	10://Clear old Data on GVL 	
		Lynus_Standards.GVL_Energy.stDataHeatingPumps[diNrOfEMS_IN_CP,diNrOfHP_OUT].bEnabled := FALSE;
			Lynus_Standards.GVL_Energy.stDataHeatingPumps[diNrOfEMS_IN_CP,diNrOfHP_OUT].arrMaxPower[1] := 0;
				Lynus_Standards.GVL_Energy.stDataHeatingPumps[diNrOfEMS_IN_CP,diNrOfHP_OUT].arrMaxPower[2] := 0;
					Lynus_Standards.GVL_Energy.stDataHeatingPumps[diNrOfEMS_IN_CP,diNrOfHP_OUT].bIsControllable := FALSE;
						Lynus_Standards.GVL_Energy.stDataHeatingPumps[diNrOfEMS_IN_CP,diNrOfHP_OUT].bIsStepSwitched := FALSE;
							Lynus_Standards.GVL_Energy.stDataHeatingPumps[diNrOfEMS_IN_CP,diNrOfHP_OUT].byErrorWarning := 0;
								Lynus_Standards.GVL_Energy.stDataHeatingPumps[diNrOfEMS_IN_CP,diNrOfHP_OUT].byNumberOfSteps := 0;
									Lynus_Standards.GVL_Energy.stDataHeatingPumps[diNrOfEMS_IN_CP,diNrOfHP_OUT].byPriority := 0;
										Lynus_Standards.GVL_Energy.stDataHeatingPumps[diNrOfEMS_IN_CP,diNrOfHP_OUT].lrElPower := 0;
											Lynus_Standards.GVL_Energy.stDataHeatingPumps[diNrOfEMS_IN_CP,diNrOfHP_OUT].lrElPowerConsumption := 0;
												Lynus_Standards.GVL_Energy.stDataHeatingPumps[diNrOfEMS_IN_CP,diNrOfHP_OUT].lrElPowerProduction := 0;
													Lynus_Standards.GVL_Energy.stDataHeatingPumps[diNrOfEMS_IN_CP,diNrOfHP_OUT].rBoilerTempHeatingSys := 0;
														Lynus_Standards.GVL_Energy.stDataHeatingPumps[diNrOfEMS_IN_CP,diNrOfHP_OUT].rBoilerTempServiceWater := 0;
															Lynus_Standards.GVL_Energy.stDataHeatingPumps[diNrOfEMS_IN_CP,diNrOfHP_OUT].rFlowTemp := 0;
																Lynus_Standards.GVL_Energy.stDataHeatingPumps[diNrOfEMS_IN_CP,diNrOfHP_OUT].rFlowTempEnergySource := 0;
																	Lynus_Standards.GVL_Energy.stDataHeatingPumps[diNrOfEMS_IN_CP,diNrOfHP_OUT].rReturnTemp := 0;
																		Lynus_Standards.GVL_Energy.stDataHeatingPumps[diNrOfEMS_IN_CP,diNrOfHP_OUT].rReturnTempEnergySource := 0;										
		diNrOfEMS_IN_CP := diNrOfEMS_IN;
			//Back to the init step
			iStateGVLData := 0;

END_CASE 	 

IF diNrOfHP_OUT > 0 AND fbNumberDevice.bNumberIsCalculatet AND diNrOfEMS_IN > 0 THEN
	Lynus_Standards.GVL_Energy.stDataHeatingPumps[diNrOfEMS_IN,diNrOfHP_OUT].bEnabled := fbHP.stDataHPOut.bEnabled;
		Lynus_Standards.GVL_Energy.stDataHeatingPumps[diNrOfEMS_IN,diNrOfHP_OUT].arrMaxPower[1] := fbHP.stDataHPOut.arrMaxPower[1];
			Lynus_Standards.GVL_Energy.stDataHeatingPumps[diNrOfEMS_IN,diNrOfHP_OUT].arrMaxPower[2] := fbHP.stDataHPOut.arrMaxPower[2];
				Lynus_Standards.GVL_Energy.stDataHeatingPumps[diNrOfEMS_IN,diNrOfHP_OUT].bIsControllable := TRUE;
					Lynus_Standards.GVL_Energy.stDataHeatingPumps[diNrOfEMS_IN,diNrOfHP_OUT].bIsStepSwitched := fbHP.stDataHPOut.bIsStepSwitched;
						Lynus_Standards.GVL_Energy.stDataHeatingPumps[diNrOfEMS_IN,diNrOfHP_OUT].byErrorWarning := fbHP.stDataHPOut.byErrorWarning;
							Lynus_Standards.GVL_Energy.stDataHeatingPumps[diNrOfEMS_IN,diNrOfHP_OUT].byNumberOfSteps := fbHP.stDataHPOut.byNumberOfSteps;
								Lynus_Standards.GVL_Energy.stDataHeatingPumps[diNrOfEMS_IN,diNrOfHP_OUT].byPriority := fbHP.stDataHPOut.byPriority;
									Lynus_Standards.GVL_Energy.stDataHeatingPumps[diNrOfEMS_IN,diNrOfHP_OUT].lrElPower := fbHP.stDataHPOut.lrElPower;
										Lynus_Standards.GVL_Energy.stDataHeatingPumps[diNrOfEMS_IN,diNrOfHP_OUT].lrElPowerConsumption := fbHP.stDataHPOut.lrElPowerConsumption;
											Lynus_Standards.GVL_Energy.stDataHeatingPumps[diNrOfEMS_IN,diNrOfHP_OUT].lrElPowerProduction := fbHP.stDataHPOut.lrElPowerProduction;
												Lynus_Standards.GVL_Energy.stDataHeatingPumps[diNrOfEMS_IN,diNrOfHP_OUT].rBoilerTempHeatingSys := fbHP.stDataHPOut.rBoilerTempHeatingSys;
													Lynus_Standards.GVL_Energy.stDataHeatingPumps[diNrOfEMS_IN,diNrOfHP_OUT].rBoilerTempServiceWater := fbHP.stDataHPOut.rBoilerTempServiceWater;
														Lynus_Standards.GVL_Energy.stDataHeatingPumps[diNrOfEMS_IN,diNrOfHP_OUT].rFlowTemp := fbHP.stDataHPOut.rFlowTemp;
															Lynus_Standards.GVL_Energy.stDataHeatingPumps[diNrOfEMS_IN,diNrOfHP_OUT].rFlowTempEnergySource := fbHP.stDataHPOut.rFlowTempEnergySource;
																Lynus_Standards.GVL_Energy.stDataHeatingPumps[diNrOfEMS_IN,diNrOfHP_OUT].rReturnTemp := fbHP.stDataHPOut.rReturnTemp;
																	Lynus_Standards.GVL_Energy.stDataHeatingPumps[diNrOfEMS_IN,diNrOfHP_OUT].rReturnTempEnergySource := fbHP.stDataHPOut.rReturnTempEnergySource;	
END_IF

(*----------------------------------------------------------Save persistent data----------------------------------------------------------------*)

arrPD[1](lrValue:= BOOL_TO_LREAL(bEnable), bEventBasedActive=> );
arrPD[2](lrValue:= BOOL_TO_LREAL(bPowerDataInvers), bEventBasedActive=> );
arrPD[3](lrValue:= DINT_TO_LREAL(diNrOfEMS_IN), bEventBasedActive=> );
arrPD[4](lrValue:= DINT_TO_LREAL(diNrOfEM_IN_HP), bEventBasedActive=> );
arrPD[5](lrValue:= DINT_TO_LREAL(diNrOfEMS_IN_CP), bEventBasedActive=> );
arrPD[6](lrValue:= REAL_TO_LREAL(stSetupHP.rMaxPower1), bEventBasedActive=> );
arrPD[7](lrValue:= REAL_TO_LREAL(stSetupHP.rMaxPower2), bEventBasedActive=> );
arrPD[8](lrValue:= BOOL_TO_LREAL(stSetupHP.bManualyOn), bEventBasedActive=> );
arrPD[9](lrValue:= BOOL_TO_LREAL(stSetupHP.bOnEmergPowerOff), bEventBasedActive=> );
arrPD[10](lrValue:= BOOL_TO_LREAL(stSetupHP.bOnEmergPowerOff), bEventBasedActive=> );
arrPD[11](lrValue:= BOOL_TO_LREAL(stSetupHP.bTimeEnabled), bEventBasedActive=> );
arrPD[12](lrValue:= BYTE_TO_LREAL(stSetupHP.byDisableSOC), bEventBasedActive=> );
arrPD[13](lrValue:= BYTE_TO_LREAL(stSetupHP.byEnableSOC), bEventBasedActive=> );
arrPD[14](lrValue:= BYTE_TO_LREAL(stSetupHP.byHourOff), bEventBasedActive=> );
arrPD[15](lrValue:= BYTE_TO_LREAL(stSetupHP.byHourOn), bEventBasedActive=> );
arrPD[16](lrValue:= BYTE_TO_LREAL(stSetupHP.byManualyTargetPower), bEventBasedActive=> );
arrPD[17](lrValue:= BYTE_TO_LREAL(stSetupHP.byMinutesOff), bEventBasedActive=> );
arrPD[18](lrValue:= BYTE_TO_LREAL(stSetupHP.byMinutesOn), bEventBasedActive=> );
arrPD[19](lrValue:= BYTE_TO_LREAL(stSetupHP.byPriority), bEventBasedActive=> );
arrPD[20](lrValue:= BYTE_TO_LREAL(stSetupHP.byTimeEnabledTargetPower), bEventBasedActive=> );
arrPD[21](lrValue:= BOOL_TO_LREAL(bNoLinear), bEventBasedActive=> );
arrPD[22](lrValue:= REAL_TO_LREAL(arrTableOfInterpolationPoints[1]), bEventBasedActive=> );
arrPD[23](lrValue:= REAL_TO_LREAL(arrTableOfInterpolationPoints[2]), bEventBasedActive=> );
arrPD[24](lrValue:= REAL_TO_LREAL(arrTableOfInterpolationPoints[3]), bEventBasedActive=> );
arrPD[25](lrValue:= REAL_TO_LREAL(arrTableOfInterpolationPoints[4]), bEventBasedActive=> );
arrPD[26](lrValue:= REAL_TO_LREAL(arrTableOfInterpolationPoints[5]), bEventBasedActive=> );
arrPD[27](lrValue:= REAL_TO_LREAL(arrTableOfInterpolationPoints[6]), bEventBasedActive=> );
arrPD[28](lrValue:= REAL_TO_LREAL(arrTableOfInterpolationPoints[7]), bEventBasedActive=> );
arrPD[29](lrValue:= REAL_TO_LREAL(arrTableOfInterpolationPoints[8]), bEventBasedActive=> );
arrPD[30](lrValue:= REAL_TO_LREAL(arrTableOfInterpolationPoints[9]), bEventBasedActive=> );
arrPD[31](lrValue:= REAL_TO_LREAL(arrTableOfInterpolationPoints[10]), bEventBasedActive=> );

END_FUNCTION_BLOCK

// ---- FBs/Heating Pump/SG Ready General/FB_HP_SGReady_General_2Stage.TcPOU
FUNCTION_BLOCK FB_HP_SGReady_General_2Stage
VAR_INPUT PERSISTENT
	bEnable									: BOOL;												//{#lynus.ag#()} //Enable the Fuctionblock and his logic
	bPowerDataInvers						: BOOL;												//With True its possible to invert all received power data from the electric meter
	diNrOfEMS_IN							: DINT;												//Number of EMS what control this Device.
	diNrOfEM_IN_HP							: DINT;												//Number of the electric meter for incoming power data. (Power Data for this Device)
	stSetupHP								: ST_Setup_HP;										//{#lynus.ag#()} //Setup heating pump
END_VAR
VAR_INPUT
END_VAR
VAR_OUTPUT
	stDataHP								: ST_HP_Output;										//{#lynus.ag#()} //Output Data Heating pump
	diNrOfHP_OUT							: DINT;												//Active Number from the heating pump for using on other functions	
	rTargetPowerForExtFunc					: REAL;												//Target Power from 0% to +100% to use on a external Function	
END_VAR
VAR
	{attribute 'hide'}
	fbHP									: FB_HeatingPump;									//Function block for heating pump
	{attribute 'hide'}
	fbNumberDevice							: FB_NumberOfDevice;								//Function block to calcualte the number of the Device
	fbDIExternalLock						: FB_XL1XXX_DI;										//Digital Input from external loock signal
	fbDIErrorHP								: FB_XL1XXX_DI;										//Digital Input for error from the heating pump
	fbDOSGReady1							: FB_XL2XXX_DO;										//1 Digital Output signal for SG Ready 
	fbDOSGReady2							: FB_XL2XXX_DO;										//2 Digital Output signal for SG Ready 
	{attribute 'hide'}
	timDissableFunctions					: TON;												//Timer to dissable the Function after Lynus_Standards.Constants_General.tTimeDissableLynusFunctions Days without connection to the Lynus Cloud
	{attribute 'hide'}
	timResetConnectionOnGVL					: TON;												//Timer to try reset the connection Flag on the GVL. (When somebody delete the Connection Function and make only a onlinechange)
	{attribute 'hide'}
	timGetTime								: TON;												//Timer to activate the function tho read out the windows system time
	{attribute 'hide'}
	FNReset									: F_TRIG;											//Internal negative edge
	{attribute 'hide'}
	fbGetSystemTime							: NT_GetTime;										//Function to read out the windows system time on the local plc
	{attribute 'hide'}
	arrPD									: ARRAY[1..20] OF FB_PersistentData_Number;			//Function to save persistent data
	{attribute 'hide'}
	byWaitInStep							: BYTE;												//Wait in Step before start to clean data on PLC
	{attribute 'hide'}
	iStateGVLData							: INT;												//State machine to handle the data on the GVL
	{attribute 'hide'}
	diNumberOfActiveBatterys				: DINT;												//Number of active batterys
	{attribute 'hide'}
	diNumberOfBatteryInverterInEPO			: DINT;												//Number of battery inverters that work in Emergency Power operation 
	{attribute 'hide'}
	diCounterForGVL							: DINT;												//Counter to clean old data on GVL
	{attribute 'hide'}
	diLPForGVL								: DINT;												//Loop to clean old data on GVL
	{attribute 'hide'}	
	dwSumSOC								: DWORD;											//Sum of the SOC from all batterys
	{attribute 'hide'}
	lrGridPower								: LREAL;											//Grid power in kW
	{attribute 'hide'}
	lrSizeGridConnection					: LREAL;											//Size of the complete grid connection
	{attribute 'hide'}
	liLPBatteryData							: LINT;												//Loop to check some data from batterys
	{attribute 'hide'}
	liLPInEPO								: LINT;												//Loop to check if 1 or more battery inverters build a island grid	
	{attribute 'hide'}
	liLPGridData							: LINT;												//Loop to check some grid data
END_VAR
VAR PERSISTENT
	{attribute 'conditionalshow'}
	diNrOfEMS_IN_CP							: DINT;												//Number of EMS what control this Device to compare with the original
END_VAR

//Creator : Kai Ebensperger
//Company : Lynus AG
//Date : 19.05.2021
//Version : 1.0.0.0

//With this function block its possible to control a Heating pump with the standard and general SG-Read Interface.
//SG-Ready are 2 Digital output signals to control the Heating pump in 4 modes.
//With this Function block is also possible to display the electric and thermal power from the heating pump
//Only 2-stage machines can be controlled with this FB.

//NOTE for diNr.....Designation => 
//_IN = Here Data come in from other Functions or go out to other functions about the GVL
//_OUT = Here Data go out to other functions about the GVL

(*------------------------------------------------------------Limits----------------------------------------------------------------------------------*)

diNrOfEMS_IN := LIMIT(0,diNrOfEMS_IN,Constants_Energy.diMaxNumberOfEMS);
	diNrOfEM_IN_HP := LIMIT(0,diNrOfEM_IN_HP,Constants_Energy.diMaxNumberOfElectricMeters);
			
(*------------------------------------------------------------------Power Data----------------------------------------------------------------------------*)

IF NOT bPowerDataInvers THEN
	fbHP.lrCounterEnergyT1_Consumption := Lynus_Standards.GVL_Energy.stDataElectricMeters[diNrOfEM_IN_HP].lrCounterEnergyT1_Production * 1000;
	fbHP.lrCounterEnergyT2_Consumption := Lynus_Standards.GVL_Energy.stDataElectricMeters[diNrOfEM_IN_HP].lrCounterEnergyT2_Production * 1000;
	fbHP.lrCounterEnergyT1_Production := Lynus_Standards.GVL_Energy.stDataElectricMeters[diNrOfEM_IN_HP].lrCounterEnergyT1_Consumption * 1000;
	fbHP.lrCounterEnergyT2_Production := Lynus_Standards.GVL_Energy.stDataElectricMeters[diNrOfEM_IN_HP].lrCounterEnergyT1_Consumption * 1000;
	fbHP.lrTotalCounterEnergy_Consumption := Lynus_Standards.GVL_Energy.stDataElectricMeters[diNrOfEM_IN_HP].lrTotalCounterEnergy_Production * 1000;
	fbHP.lrTotalCounterEnergy_Production := Lynus_Standards.GVL_Energy.stDataElectricMeters[diNrOfEM_IN_HP].lrTotalCounterEnergy_Consumption * 1000;
		fbHP.lrElPowerHP := (Lynus_Standards.GVL_Energy.stDataElectricMeters[diNrOfEM_IN_HP].lrPower * 1000) * - 1;
ELSE
	fbHP.lrCounterEnergyT1_Consumption := Lynus_Standards.GVL_Energy.stDataElectricMeters[diNrOfEM_IN_HP].lrCounterEnergyT1_Consumption * 1000;
	fbHP.lrCounterEnergyT2_Consumption := Lynus_Standards.GVL_Energy.stDataElectricMeters[diNrOfEM_IN_HP].lrCounterEnergyT2_Consumption * 1000;
	fbHP.lrCounterEnergyT1_Production := Lynus_Standards.GVL_Energy.stDataElectricMeters[diNrOfEM_IN_HP].lrCounterEnergyT1_Production * 1000;
	fbHP.lrCounterEnergyT2_Production := Lynus_Standards.GVL_Energy.stDataElectricMeters[diNrOfEM_IN_HP].lrCounterEnergyT2_Production * 1000;
	fbHP.lrTotalCounterEnergy_Consumption := Lynus_Standards.GVL_Energy.stDataElectricMeters[diNrOfEM_IN_HP].lrTotalCounterEnergy_Consumption * 1000;
	fbHP.lrTotalCounterEnergy_Production := Lynus_Standards.GVL_Energy.stDataElectricMeters[diNrOfEM_IN_HP].lrTotalCounterEnergy_Production * 1000;
		fbHP.lrElPowerHP := Lynus_Standards.GVL_Energy.stDataElectricMeters[diNrOfEM_IN_HP].lrPower * 1000;
END_IF

(*-------------------------------------------------------------Calcualte the number of HP---------------------------------------------------------------*)

fbNumberDevice(
	diActualNumberOfDevices:= Lynus_Standards.GVL_Energy.stNumberOfDevices.diNumberOfHP, 
	diMaxNumberOfDevices:= Constants_Energy.diMaxNumberOfHeatingPumps, 
	udiCounterOnlineChange:= TwinCAT_SystemInfoVarList._AppInfo.OnlineChangeCnt, 
	bNumberIsCalculatet=> , 
	bFPNumberIsCalculatet=> , 
	bOnlineChange=> , 
	diNumberForThisDevice=> diNrOfHP_OUT, 
	diNumberOfTotalDevices=> );

//Write new Numer on GVL
IF fbNumberDevice.bFPNumberIsCalculatet THEN
	Lynus_Standards.GVL_Energy.stNumberOfDevices.diNumberOfHP := fbNumberDevice.diNumberOfTotalDevices;	
END_IF 

//Delete old Number on GVL
IF fbNumberDevice.bOnlineChange THEN 
	Lynus_Standards.GVL_Energy.stNumberOfDevices.diNumberOfHP := diNrOfHP_OUT;	
		iStateGVLData := 1; 
END_IF

(*-------------------------------------------------------------Get the local windows system time for this plc---------------------------------------------------------------*)
timGetTime(IN:= bEnable AND NOT timGetTime.Q, PT:= T#30S, Q=> , ET=> );

fbGetSystemTime(
	NETID:= , 
	START:= timGetTime.Q AND NOT fbGetSystemTime.BUSY, 
	TMOUT:= , 
	BUSY=> , 
	ERR=> , 
	ERRID=> , 
	TIMESTR=> );	

fbHP.stSystemTime.wHour := fbGetSystemTime.TIMESTR.wHour;
	fbHP.stSystemTime.wMinute := fbGetSystemTime.TIMESTR.wMinute;	

(*-------------------------------------------------------------Service from Backend is ready and check the connection to backen for dissabel/enable Function---------------------------------------------------------------*)

//Try to reset the variable for connection on the GVL. When all is normal then the Lynus Mqtt connection function set this variable to true in the next cycle
//When we have no connection to the backend then after Lynus_Standards.Constants_General.tTimeDissableLynusFunctions days the Function is dissabled with all of his functionalities
timResetConnectionOnGVL(IN:= NOT timResetConnectionOnGVL.Q, PT:= T#1H, Q=> , ET=> );
	IF timResetConnectionOnGVL.Q THEN Lynus_Standards.GVL_Communicator.bStateConnectionToEnableFunctions := FALSE; END_IF
		IF NOT Lynus_Standards.GVL_Communicator.bStateConnectionToEnableFunctions THEN timDissableFunctions.IN := TRUE; ELSE timDissableFunctions.IN := FALSE; END_IF  
			timDissableFunctions(IN:= , PT:= Lynus_Standards.Constants_General.tTimeDissableLynusFunctions, Q=> , ET=> );		
	
(*------------------------------------------------------------------Error and Reset----------------------------------------------------------------------------*)	

fbDIErrorHP(bInvers:= FALSE, bSignal=> );

IF timDissableFunctions.Q THEN fbHP.bWarning := TRUE; fbHP.iWarningCode := 0; ELSE fbHP.bWarning := FALSE; END_IF 	
	IF Lynus_Standards.GVL_Energy.stNumberOfDevices.diNumberOfHP > Constants_Energy.diMaxNumberOfHeatingPumps OR fbDIErrorHP.bSignal OR fbGetSystemTime.ERR THEN fbHP.bError := TRUE; ELSE fbHP.bError := FALSE; END_IF 

IF Lynus_Standards.GVL_Energy.stNumberOfDevices.diNumberOfHP > Constants_Energy.diMaxNumberOfHeatingPumps THEN fbHP.iErrorCode := 1;
ELSIF fbGetSystemTime.ERR THEN fbHP.iErrorCode := 2; 
ELSIF fbDIErrorHP.bSignal THEN fbHP.iErrorCode := 0;
END_IF

FNReset(CLK:= fbHP.stDataHPOut.bSReset, Q=> );

(*------------------------------------------------------------------Logic----------------------------------------------------------------------------*)

//Calcualte the total SOC if we have more then 1 battery in our system
diNumberOfActiveBatterys := 0;
	dwSumSOC := 0;
		FOR liLPBatteryData := 1 TO Constants_Energy.diMaxNumberOfBatterys BY 1 DO
			IF Lynus_Standards.GVL_Energy.stDataOfBatterys[diNrOfEMS_IN,liLPBatteryData].bEnabled THEN diNumberOfActiveBatterys := diNumberOfActiveBatterys + 1; END_IF
				dwSumSOC := dwSumSOC + Lynus_Standards.GVL_Energy.stDataOfBatterys[diNrOfEMS_IN,liLPBatteryData].dwSOC;
		END_FOR
	
IF diNumberOfActiveBatterys > 0 THEN
	fbHP.dwBatterySOC := DINT_TO_DWORD(DWORD_TO_DINT(dwSumSOC) / diNumberOfActiveBatterys);
ELSE
	fbHP.dwBatterySOC := 100;	//When we have no battery in the ems system
END_IF

//Check if one or more Batterysystems or batteryinverter make island mode
diNumberOfBatteryInverterInEPO := 0;
	FOR liLPInEPO := 1 TO Constants_Energy.diMaxNumberOfBatteryInverters BY 1 DO
		IF Lynus_Standards.GVL_Energy.stDataOfBatteryInverters[diNrOfEMS_IN,liLPInEPO].bWorkOnIslandMode THEN fbHP.bEPOIsActive := TRUE; diNumberOfBatteryInverterInEPO := diNumberOfBatteryInverterInEPO + 1; END_IF
	END_FOR 
		IF diNumberOfBatteryInverterInEPO <= 0 THEN fbHP.bEPOIsActive := FALSE; END_IF

//Check the max. power of the grid connection and the sum of grid power
lrSizeGridConnection := 0;
	lrGridPower := 0;
		FOR liLPGridData := 1 TO Constants_Energy.diMaxNumberOfGridConnections BY 1 DO
			lrSizeGridConnection := lrSizeGridConnection + Lynus_Standards.GVL_Energy.stDataGridConnections[diNrOfEMS_IN,liLPGridData].rSizeGridConn;
				lrGridPower := lrGridPower + Lynus_Standards.GVL_Energy.stDataGridConnections[diNrOfEMS_IN,liLPGridData].lrPower;
		END_FOR		

//Feedback for HP is running
IF fbHP.arrTargetPower[1] > 0 OR fbHP.arrTargetPower[2] > 0 THEN fbHP.bHPIsRunning := TRUE; ELSE fbHP.bHPIsRunning := FALSE; END_IF 
		
//Digital input for external lock signal
fbDIExternalLock(bInvers:= FALSE, bSignal=> );

//Functionblock HP
fbHP(
	bEnable:= bEnable AND NOT timDissableFunctions.Q,  
	bError:= , 
	bWarning:= , 
	bIsStepSwitched:= TRUE, 
	bEPOIsActive:= , 
	bExternalLock:= fbDIExternalLock.bSignal, 
	bReset:= FNReset.Q, 
	bExternalOnCommand:= Lynus_Standards.GVL_Energy.stDataHeatingPumps[diNrOfEMS_IN,diNrOfHP_OUT].bExternalOnCommand, 
	bWriteWithDelay:= TRUE,
	bHPIsRunning:= , 
	iErrorCode:= , 
	iWarningCode:= , 
	dwBatterySOC:= , 
	diNumberOfHP:= diNrOfHP_OUT, 
	rBoilerTempHeatingSys:= 0, 
	rBoilerTempServiceWater:= 0, 
	rFlowTemp:= 0, 
	rReturnTemp:= 0, 
	rFlowTempEnergySource:= 0, 
	rReturnTempEnergySource:= 0, 
	lrSizeGridConnection:= lrSizeGridConnection, 
	lrGridPower:= lrGridPower, 
	lrTotalCounterEnergy_Consumption:= , 
	lrTotalCounterEnergy_Production:= , 
	lrCounterEnergyT1_Consumption:= , 
	lrCounterEnergyT2_Consumption:= , 
	lrCounterEnergyT1_Production:= , 
	lrCounterEnergyT2_Production:= , 
	lrCounterThermalEnergy_Heating:= 0, 
	lrCounterThermalEnergy_Water:= 0, 
	lrElPowerHP:= , 
	arrTargetPower:= Lynus_Standards.GVL_Energy.stDataHeatingPumps[diNrOfEMS_IN,diNrOfHP_OUT].arrTargetPowerEMS, 
	tOnDelayExternalOn:= T#2M, 
	tOffDelayExternalOn:= T#2H, 
	tMinOnTime:= T#1.5H,
	tTimDelayOutput:= T#5S, 
	stSystemTime:= , 
	stSetupHP:= stSetupHP, 
	stDataHPOut=> , 
	stDataHPOutDelay=> stDataHP, 
	arrPercentValuesSteps=> );

//Target Power, to use this on a external Function
rTargetPowerForExtFunc := fbHP.stDataHPOut.rTargetPower;
	
(*-------------------------------------------------------------------------Output----------------------------------------------------------------------*)

//Operating Mode (When Manualy mode is active)
IF stSetupHP.bManualyOn THEN	
	//Operating Mode 1 SG Ready
	IF NOT fbHP.stDataHPOut.bOutput THEN 
		fbDOSGReady1.bSignal := FALSE; 
		fbDOSGReady2.bSignal := TRUE; 
	END_IF
		//Operating Mode 2 SG Ready
		IF fbHP.stDataHPOut.rTargetPower < fbHP.arrPercentValuesSteps[1] AND fbHP.stDataHPOut.rTargetPower > 0 THEN 
			fbDOSGReady1.bSignal := FALSE; 
			fbDOSGReady2.bSignal := FALSE; 
		END_IF
			//Operating Mode 3 SG Ready
			IF fbHP.stDataHPOut.rTargetPower >= fbHP.arrPercentValuesSteps[1] AND fbHP.arrPercentValuesSteps[1] > 0 THEN 
				fbDOSGReady1.bSignal := TRUE; 
				fbDOSGReady2.bSignal := FALSE;
			END_IF
				//Operating Mode 4 SG Ready	
				IF fbHP.stDataHPOut.rTargetPower >= 100 AND fbHP.stDataHPOut.byNumberOfSteps > 1 THEN 
					fbDOSGReady1.bSignal := TRUE; 
					fbDOSGReady2.bSignal := TRUE; 
				END_IF
ELSE
	//Operating Mode (When Normal mode is active) 
	//Operating Mode 1 SG Ready
	IF NOT fbHP.stDataHPOut.bOutput THEN
		fbDOSGReady1.bSignal := FALSE; 
		fbDOSGReady2.bSignal := TRUE;
	ELSE
		//Operating Mode 2 SG Ready
		IF fbHP.stDataHPOut.bOutput THEN 
			fbDOSGReady1.bSignal := FALSE; 
			fbDOSGReady2.bSignal := FALSE; 
		END_IF
			//Operating Mode 3 SG Ready
			IF fbHP.stDataHPOut.rTargetPower >= fbHP.arrPercentValuesSteps[1] AND fbHP.arrPercentValuesSteps[1] > 0 THEN 
				fbDOSGReady1.bSignal := TRUE; 
				fbDOSGReady2.bSignal := FALSE; 
			END_IF
				//Operating Mode 4 SG Ready	
				IF fbHP.stDataHPOut.rTargetPower >= 100 AND fbHP.stDataHPOut.byNumberOfSteps > 1 THEN 
					fbDOSGReady1.bSignal := TRUE; 
					fbDOSGReady2.bSignal := TRUE;
				END_IF
	END_IF	
END_IF

fbDOSGReady1(bInvers:= FALSE, bSignal:= );
	fbDOSGReady2(bInvers:= FALSE, bSignal:= );

(*-----------------------------------------------------------Handle data to Global structure for the heating pump-----------------------------------------------------------------*)

//Delte al old Data on GVL after a online change or change on the variable diNrOfEMS_IDOD
IF diNrOfEMS_IN <> diNrOfEMS_IN_CP AND iStateGVLData = 0 THEN iStateGVLData := 10; END_IF 

CASE iStateGVLData OF
	
	0://Init Step
		byWaitInStep := 0;
			diCounterForGVL := 1;
	
	1://Wait for 4 Steps before clean al Data on GVL
		byWaitInStep := byWaitInStep + 1;
			IF byWaitInStep >= 4 AND fbNumberDevice.bNumberIsCalculatet THEN iStateGVLData := 2; END_IF
				//To much Devices, back to the Init step
				IF byWaitInStep >= 4 AND NOT fbNumberDevice.bNumberIsCalculatet THEN iStateGVLData := 0; END_IF	
			
	2://Clear all Data in GVL
		FOR diLPForGVL := 1 TO Constants_Energy.diMaxNumberOfEMS BY 1 DO
			Lynus_Standards.GVL_Energy.stDataHeatingPumps[diLPForGVL,diCounterForGVL].bEnabled := FALSE;
				Lynus_Standards.GVL_Energy.stDataHeatingPumps[diLPForGVL,diCounterForGVL].arrMaxPower[1] := 0;
					Lynus_Standards.GVL_Energy.stDataHeatingPumps[diLPForGVL,diCounterForGVL].arrMaxPower[2] := 0;
						Lynus_Standards.GVL_Energy.stDataHeatingPumps[diLPForGVL,diCounterForGVL].bIsControllable := FALSE;
							Lynus_Standards.GVL_Energy.stDataHeatingPumps[diLPForGVL,diCounterForGVL].bIsStepSwitched := FALSE;
								Lynus_Standards.GVL_Energy.stDataHeatingPumps[diLPForGVL,diCounterForGVL].byErrorWarning := 0;
									Lynus_Standards.GVL_Energy.stDataHeatingPumps[diLPForGVL,diCounterForGVL].byNumberOfSteps := 0;
										Lynus_Standards.GVL_Energy.stDataHeatingPumps[diLPForGVL,diCounterForGVL].byPriority := 0;
											Lynus_Standards.GVL_Energy.stDataHeatingPumps[diLPForGVL,diCounterForGVL].lrElPower := 0;
												Lynus_Standards.GVL_Energy.stDataHeatingPumps[diLPForGVL,diCounterForGVL].lrElPowerConsumption := 0;
													Lynus_Standards.GVL_Energy.stDataHeatingPumps[diLPForGVL,diCounterForGVL].lrElPowerProduction := 0;
														Lynus_Standards.GVL_Energy.stDataHeatingPumps[diLPForGVL,diCounterForGVL].rBoilerTempHeatingSys := 0;
															Lynus_Standards.GVL_Energy.stDataHeatingPumps[diLPForGVL,diCounterForGVL].rBoilerTempServiceWater := 0;
																Lynus_Standards.GVL_Energy.stDataHeatingPumps[diLPForGVL,diCounterForGVL].rFlowTemp := 0;
																	Lynus_Standards.GVL_Energy.stDataHeatingPumps[diLPForGVL,diCounterForGVL].rFlowTempEnergySource := 0;
																		Lynus_Standards.GVL_Energy.stDataHeatingPumps[diLPForGVL,diCounterForGVL].rReturnTemp := 0;
																			Lynus_Standards.GVL_Energy.stDataHeatingPumps[diLPForGVL,diCounterForGVL].rReturnTempEnergySource := 0;
																				//Set also the target value from ems back here to 0 and not in EMS function because EMS is in Standy when we have a online change (Problem when we delete a ems function and make a online change)
																				Lynus_Standards.GVL_Energy.stDataHeatingPumps[diLPForGVL,diCounterForGVL].arrTargetPowerEMS[1] := 0;
																					Lynus_Standards.GVL_Energy.stDataHeatingPumps[diLPForGVL,diCounterForGVL].arrTargetPowerEMS[2] := 0;
																						Lynus_Standards.GVL_Energy.stDataHeatingPumps[diLPForGVL,diCounterForGVL].bExternalOnCommand := FALSE;	
		END_FOR
			diCounterForGVL := diCounterForGVL + 1;
				diCounterForGVL := LIMIT(0,diCounterForGVL,Constants_Energy.diMaxNumberOfHeatingPumps);
					//Back to the init step
					IF diCounterForGVL >= Constants_Energy.diMaxNumberOfHeatingPumps THEN iStateGVLData := 0; END_IF

	10://Clear old Data on GVL 	
		Lynus_Standards.GVL_Energy.stDataHeatingPumps[diNrOfEMS_IN_CP,diNrOfHP_OUT].bEnabled := FALSE;
			Lynus_Standards.GVL_Energy.stDataHeatingPumps[diNrOfEMS_IN_CP,diNrOfHP_OUT].arrMaxPower[1] := 0;
				Lynus_Standards.GVL_Energy.stDataHeatingPumps[diNrOfEMS_IN_CP,diNrOfHP_OUT].arrMaxPower[2] := 0;
					Lynus_Standards.GVL_Energy.stDataHeatingPumps[diNrOfEMS_IN_CP,diNrOfHP_OUT].bIsControllable := FALSE;
						Lynus_Standards.GVL_Energy.stDataHeatingPumps[diNrOfEMS_IN_CP,diNrOfHP_OUT].bIsStepSwitched := FALSE;
							Lynus_Standards.GVL_Energy.stDataHeatingPumps[diNrOfEMS_IN_CP,diNrOfHP_OUT].byErrorWarning := 0;
								Lynus_Standards.GVL_Energy.stDataHeatingPumps[diNrOfEMS_IN_CP,diNrOfHP_OUT].byNumberOfSteps := 0;
									Lynus_Standards.GVL_Energy.stDataHeatingPumps[diNrOfEMS_IN_CP,diNrOfHP_OUT].byPriority := 0;
										Lynus_Standards.GVL_Energy.stDataHeatingPumps[diNrOfEMS_IN_CP,diNrOfHP_OUT].lrElPower := 0;
											Lynus_Standards.GVL_Energy.stDataHeatingPumps[diNrOfEMS_IN_CP,diNrOfHP_OUT].lrElPowerConsumption := 0;
												Lynus_Standards.GVL_Energy.stDataHeatingPumps[diNrOfEMS_IN_CP,diNrOfHP_OUT].lrElPowerProduction := 0;
													Lynus_Standards.GVL_Energy.stDataHeatingPumps[diNrOfEMS_IN_CP,diNrOfHP_OUT].rBoilerTempHeatingSys := 0;
														Lynus_Standards.GVL_Energy.stDataHeatingPumps[diNrOfEMS_IN_CP,diNrOfHP_OUT].rBoilerTempServiceWater := 0;
															Lynus_Standards.GVL_Energy.stDataHeatingPumps[diNrOfEMS_IN_CP,diNrOfHP_OUT].rFlowTemp := 0;
																Lynus_Standards.GVL_Energy.stDataHeatingPumps[diNrOfEMS_IN_CP,diNrOfHP_OUT].rFlowTempEnergySource := 0;
																	Lynus_Standards.GVL_Energy.stDataHeatingPumps[diNrOfEMS_IN_CP,diNrOfHP_OUT].rReturnTemp := 0;
																		Lynus_Standards.GVL_Energy.stDataHeatingPumps[diNrOfEMS_IN_CP,diNrOfHP_OUT].rReturnTempEnergySource := 0;										
		diNrOfEMS_IN_CP := diNrOfEMS_IN;
			//Back to the init step
			iStateGVLData := 0;

END_CASE 	 

IF diNrOfHP_OUT > 0 AND fbNumberDevice.bNumberIsCalculatet AND diNrOfEMS_IN > 0 THEN
	Lynus_Standards.GVL_Energy.stDataHeatingPumps[diNrOfEMS_IN,diNrOfHP_OUT].bEnabled := fbHP.stDataHPOut.bEnabled;
		Lynus_Standards.GVL_Energy.stDataHeatingPumps[diNrOfEMS_IN,diNrOfHP_OUT].arrMaxPower[1] := fbHP.stDataHPOut.arrMaxPower[1];
			Lynus_Standards.GVL_Energy.stDataHeatingPumps[diNrOfEMS_IN,diNrOfHP_OUT].arrMaxPower[2] := fbHP.stDataHPOut.arrMaxPower[2];
				Lynus_Standards.GVL_Energy.stDataHeatingPumps[diNrOfEMS_IN,diNrOfHP_OUT].bIsControllable := TRUE;
					Lynus_Standards.GVL_Energy.stDataHeatingPumps[diNrOfEMS_IN,diNrOfHP_OUT].bIsStepSwitched := fbHP.stDataHPOut.bIsStepSwitched;
						Lynus_Standards.GVL_Energy.stDataHeatingPumps[diNrOfEMS_IN,diNrOfHP_OUT].byErrorWarning := fbHP.stDataHPOut.byErrorWarning;
							Lynus_Standards.GVL_Energy.stDataHeatingPumps[diNrOfEMS_IN,diNrOfHP_OUT].byNumberOfSteps := fbHP.stDataHPOut.byNumberOfSteps;
								Lynus_Standards.GVL_Energy.stDataHeatingPumps[diNrOfEMS_IN,diNrOfHP_OUT].byPriority := fbHP.stDataHPOut.byPriority;
									Lynus_Standards.GVL_Energy.stDataHeatingPumps[diNrOfEMS_IN,diNrOfHP_OUT].lrElPower := fbHP.stDataHPOut.lrElPower;
										Lynus_Standards.GVL_Energy.stDataHeatingPumps[diNrOfEMS_IN,diNrOfHP_OUT].lrElPowerConsumption := fbHP.stDataHPOut.lrElPowerConsumption;
											Lynus_Standards.GVL_Energy.stDataHeatingPumps[diNrOfEMS_IN,diNrOfHP_OUT].lrElPowerProduction := fbHP.stDataHPOut.lrElPowerProduction;
												Lynus_Standards.GVL_Energy.stDataHeatingPumps[diNrOfEMS_IN,diNrOfHP_OUT].rBoilerTempHeatingSys := fbHP.stDataHPOut.rBoilerTempHeatingSys;
													Lynus_Standards.GVL_Energy.stDataHeatingPumps[diNrOfEMS_IN,diNrOfHP_OUT].rBoilerTempServiceWater := fbHP.stDataHPOut.rBoilerTempServiceWater;
														Lynus_Standards.GVL_Energy.stDataHeatingPumps[diNrOfEMS_IN,diNrOfHP_OUT].rFlowTemp := fbHP.stDataHPOut.rFlowTemp;
															Lynus_Standards.GVL_Energy.stDataHeatingPumps[diNrOfEMS_IN,diNrOfHP_OUT].rFlowTempEnergySource := fbHP.stDataHPOut.rFlowTempEnergySource;
																Lynus_Standards.GVL_Energy.stDataHeatingPumps[diNrOfEMS_IN,diNrOfHP_OUT].rReturnTemp := fbHP.stDataHPOut.rReturnTemp;
																	Lynus_Standards.GVL_Energy.stDataHeatingPumps[diNrOfEMS_IN,diNrOfHP_OUT].rReturnTempEnergySource := fbHP.stDataHPOut.rReturnTempEnergySource;	
END_IF

(*----------------------------------------------------------Save persistent data----------------------------------------------------------------*)

arrPD[1](lrValue:= BOOL_TO_LREAL(bEnable), bEventBasedActive=> );
arrPD[2](lrValue:= BOOL_TO_LREAL(bPowerDataInvers), bEventBasedActive=> );
arrPD[3](lrValue:= DINT_TO_LREAL(diNrOfEMS_IN), bEventBasedActive=> );
arrPD[4](lrValue:= DINT_TO_LREAL(diNrOfEM_IN_HP), bEventBasedActive=> );
arrPD[5](lrValue:= DINT_TO_LREAL(diNrOfEMS_IN_CP), bEventBasedActive=> );
arrPD[6](lrValue:= REAL_TO_LREAL(stSetupHP.rMaxPower1), bEventBasedActive=> );
arrPD[7](lrValue:= REAL_TO_LREAL(stSetupHP.rMaxPower2), bEventBasedActive=> );
arrPD[8](lrValue:= BOOL_TO_LREAL(stSetupHP.bManualyOn), bEventBasedActive=> );
arrPD[9](lrValue:= BOOL_TO_LREAL(stSetupHP.bOnEmergPowerOff), bEventBasedActive=> );
arrPD[10](lrValue:= BOOL_TO_LREAL(stSetupHP.bOnEmergPowerOff), bEventBasedActive=> );
arrPD[11](lrValue:= BOOL_TO_LREAL(stSetupHP.bTimeEnabled), bEventBasedActive=> );
arrPD[12](lrValue:= BYTE_TO_LREAL(stSetupHP.byDisableSOC), bEventBasedActive=> );
arrPD[13](lrValue:= BYTE_TO_LREAL(stSetupHP.byEnableSOC), bEventBasedActive=> );
arrPD[14](lrValue:= BYTE_TO_LREAL(stSetupHP.byHourOff), bEventBasedActive=> );
arrPD[15](lrValue:= BYTE_TO_LREAL(stSetupHP.byHourOn), bEventBasedActive=> );
arrPD[16](lrValue:= BYTE_TO_LREAL(stSetupHP.byManualyTargetPower), bEventBasedActive=> );
arrPD[17](lrValue:= BYTE_TO_LREAL(stSetupHP.byMinutesOff), bEventBasedActive=> );
arrPD[18](lrValue:= BYTE_TO_LREAL(stSetupHP.byMinutesOn), bEventBasedActive=> );
arrPD[19](lrValue:= BYTE_TO_LREAL(stSetupHP.byPriority), bEventBasedActive=> );
arrPD[20](lrValue:= BYTE_TO_LREAL(stSetupHP.byTimeEnabledTargetPower), bEventBasedActive=> );

END_FUNCTION_BLOCK

// ---- FBs/House Consumption/Virtual/FB_HouseC_Power_Virtual.TcPOU
FUNCTION_BLOCK FB_HouseC_Power_Virtual
VAR_INPUT PERSISTENT
	bEnable									: BOOL;													//{#lynus.ag#()} //Enable the Fuctionblock and his logic
	diNrOfEMS_IN							: DINT;													//Number of EMS from what this Device received Data
END_VAR
VAR_INPUT
	bSetDefault								: BOOL;													//With this Input can set the default Value from the Counter from the Input to the Counter at the Output									
	lrCounterConsumptionSetDefault			: LREAL;												//Set Default value for Consumption Counter
	lrCounterProductionSetDefault			: LREAL;												//Set Default value for Production Counter
END_VAR
VAR_OUTPUT
	stDataHouseC							: ST_HouseConsumption_Output;							//{#lynus.ag#()} //House consumption output data
	diNrOfHouseC_OUT						: DINT;													//Active Number from the House connection for using on other functions
END_VAR
VAR
	{attribute 'hide'}
	fbHouseC								: FB_HouseConsumption;									//Function for House consumption
	{attribute 'hide'}
	fbNumberDevice							: FB_NumberOfDevice;									//Function block to calcualte the number of the Device
	{attribute 'hide'}
	TaskIndex								: GETCURTASKINDEX;										//Function to read out the task index	
	{attribute 'hide'}
	timSaveCSProd							: TON;													//Timer to save the Counter Status from production on persistent data
	{attribute 'hide'}
	timSaveCSCons							: TON;													//Timer to save the Counter Status from Consumption on persistent data
	{attribute 'hide'}
	timDissableFunctions					: TON;													//Timer to dissable the Function after Lynus_Standards.Constants_General.tTimeDissableLynusFunctions Days without connection to the Lynus Cloud
	{attribute 'hide'}
	timResetConnectionOnGVL					: TON;													//Timer to try reset the connection Flag on the GVL. (When somebody delete the Connection Function and make only a onlinechange)
	{attribute 'hide'}
	FPSetDefault							: R_TRIG;												//Internal positive Edge
	{attribute 'hide'}
	arrPD									: ARRAY[1..4] OF FB_PersistentData_Number;				//Function to save persistent data 
	{attribute 'hide'}
	bError									: BOOL;													//Error from external Devices
	{attribute 'hide'}
	byWaitInStep							: BYTE;													//Wait in Step before start to clean data on PLC
	{attribute 'hide'}
	iStateGVLData							: INT;													//State machine to handle the data on the GVL
	{attribute 'hide'}
	diCounterForGVL							: DINT;													//Counter to clean old data on GVL
	{attribute 'hide'}
	udicycleTime							: UDINT;												//Cycletime of plc
	{attribute 'hide'}
	lrPowerProduction						: LREAL;												//Complete Power Production from al Devices of this EMS in kW 
	{attribute 'hide'}
	lrPowerBattery							: LREAL;												//Complete Battery Power from al Batterys of this EMS in kW 
	{attribute 'hide'}
	lrPowerGrid								: LREAL;												//Complete Grid Power from al Grids of this EMS in kW 
	{attribute 'hide'}
	lrCounterConsumption_CP					: LREAL;												//Counter Status Consumption with Unit kW/h to compare for save persistent
	{attribute 'hide'}
	lrCounterProduction_CP					: LREAL;												//Counter Status Production with Unit kW/h to compare for save persistent
	{attribute 'hide'}
	lrTotalPower							: LREAL;												//Total power with unit kW
	{attribute 'hide'}
	lrTotalPower_CP							: LREAL;												//Total power with unit kW to trigger the calculation for energy
	{attribute 'hide'}
	lrCyclesForMinute						: LREAL;												//Cycles what the plc need for 1 minute 
	{attribute 'hide'}
	lrPastTime								: LREAL;												//Past time in hours 
	{attribute 'hide'}
	lrSumToCalculate						: LREAL;												//Actual sum of the energy counters before start the calculation with unit kW/h
	{attribute 'hide'}
	liLPPower								: LINT;													//Loop to calculate the total power
END_VAR
VAR PERSISTENT
	{attribute 'conditionalshow'}
	lrCounterConsumption					: LREAL;												//Counter Status Consumption with Unit kW/h
	{attribute 'conditionalshow'}
	lrCounterProduction						: LREAL;												//Counter Status Production with Unit kW/h
END_VAR

//Creator : Kai Ebensperger
//Company : Lynus AG
//Date : 15.06.2021
//Version : 1.0.0.0

//With this function block its possible to show the power data from a house.
//The power data in this function block is calculated by all the other consumers and producers. So the output data is not messured.
//Use only one of this Function block per each EMS
//NOTE : The output from this Function Block is not 100% perfect why the value is only calculatet and not messured.

//NOTE for diNr.....Designation => 
//_IN = Here Data come in from other Functions or go out to other functions about the GVL
//_OUT = Here Data go out to other functions about the GVL

(*------------------------------------------------------------Limits----------------------------------------------------------------------------------*)

diNrOfEMS_IN := LIMIT(0,diNrOfEMS_IN,Constants_Energy.diMaxNumberOfEMS);

(*-------------------------------------------------------------Calcualte the number of House Consumption---------------------------------------------------------------*)

fbNumberDevice(
	diActualNumberOfDevices:= Lynus_Standards.GVL_Energy.stNumberOfDevices.diNumberOfHouseConsumption, 
	diMaxNumberOfDevices:= Constants_Energy.diMaxNumberOfHouseConsumptions, 
	udiCounterOnlineChange:= TwinCAT_SystemInfoVarList._AppInfo.OnlineChangeCnt, 
	bNumberIsCalculatet=> , 
	bFPNumberIsCalculatet=> , 
	bOnlineChange=> , 
	diNumberForThisDevice=> diNrOfHouseC_OUT, 
	diNumberOfTotalDevices=> );

//Write new Numer on GVL
IF fbNumberDevice.bFPNumberIsCalculatet THEN
	Lynus_Standards.GVL_Energy.stNumberOfDevices.diNumberOfHouseConsumption := fbNumberDevice.diNumberOfTotalDevices;	
END_IF 

//Delete old Number on GVL
IF fbNumberDevice.bOnlineChange THEN 
	Lynus_Standards.GVL_Energy.stNumberOfDevices.diNumberOfHouseConsumption := diNrOfHouseC_OUT;	
		iStateGVLData := 1; 
END_IF

(*-------------------------------------------------------------Calcualte the power of the house---------------------------------------------------------------*)	

lrPowerProduction := 0;
	lrPowerBattery := 0;
		lrPowerGrid := 0;
			bError := FALSE;

//Batterypower
FOR liLPPower := 1 TO Constants_Energy.diMaxNumberOfBatterys BY 1 DO
	lrPowerBattery := lrPowerBattery + Lynus_Standards.GVL_Energy.stDataOfBatterys[diNrOfEMS_IN,liLPPower].lrPower;	
		IF Lynus_Standards.GVL_Energy.stDataOfBatterys[diNrOfEMS_IN,liLPPower].byErrorWarning = 2 THEN bError := TRUE; END_IF 
END_FOR 
 	//Generator power
	FOR liLPPower := 1 TO Constants_Energy.diMaxNumberOfGenerators BY 1 DO
		lrPowerProduction := lrPowerProduction + Lynus_Standards.GVL_Energy.stDataOfGenerators[liLPPower].lrPowerProduction;	
			IF Lynus_Standards.GVL_Energy.stDataOfGenerators[liLPPower].byErrorWarning = 2 THEN bError := TRUE; END_IF		
	END_FOR 
		//PV power
		FOR liLPPower := 1 TO Constants_Energy.diMaxNumberOfPvSystems BY 1 DO
			lrPowerProduction := lrPowerProduction + Lynus_Standards.GVL_Energy.stDataOfPvSystems[liLPPower].lrPowerProduction;	
				IF Lynus_Standards.GVL_Energy.stDataOfPvSystems[liLPPower].byErrorWarning = 2 THEN bError := TRUE; END_IF		
		END_FOR	
			//Grid power	
			FOR liLPPower := 1 TO Constants_Energy.diMaxNumberOfGridConnections BY 1 DO
				lrPowerGrid := lrPowerGrid + Lynus_Standards.GVL_Energy.stDataGridConnections[diNrOfEMS_IN,liLPPower].lrPower;	
					IF Lynus_Standards.GVL_Energy.stDataGridConnections[diNrOfEMS_IN,liLPPower].byErrorWarning = 2 THEN bError := TRUE; END_IF 
			END_FOR 

//Complete power
lrTotalPower := lrPowerProduction + lrPowerGrid + lrPowerBattery;
	lrTotalPower := LIMIT(0,lrTotalPower,100000);							

(*-------------------------------------------------------------Calcualte the energy of the house---------------------------------------------------------------*)
							
//Read out the Taskindex
TaskIndex(index=> );							

//Set default Value
FPSetDefault(CLK:= bSetDefault, Q=> );
	IF FPSetDefault.Q THEN 
		lrCounterConsumption_CP := lrCounterConsumptionSetDefault;
			lrCounterProduction_CP := lrCounterProductionSetDefault;
	END_IF
						
//Save the persistent counter status to the counter status for compare on the first plc cycle	
IF TwinCAT_SystemInfoVarList._TaskInfo[TaskIndex.index].FirstCycle THEN 
	lrCounterConsumption_CP := lrCounterConsumption;
		lrCounterProduction_CP := lrCounterProduction;
END_IF											

//Timer to save the Energy Counters persistent every 12 hours											
timSaveCSProd(IN:= lrCounterProduction <> lrCounterProduction_CP, PT:= T#12H, Q=> , ET=> );
	timSaveCSCons(IN:= lrCounterConsumption <> lrCounterConsumption_CP, PT:= T#12H, Q=> , ET=> );

IF timSaveCSProd.Q THEN lrCounterProduction := lrCounterProduction_CP; END_IF 
	IF timSaveCSCons.Q THEN lrCounterConsumption := lrCounterConsumption_CP; END_IF  
	
//Write Data when the Event Based saving on persitent Data is not active
IF NOT arrPD[3].bEventBasedActive AND NOT arrPD[4].bEventBasedActive THEN
	lrCounterProduction := lrCounterProduction_CP;
		lrCounterConsumption := lrCounterConsumption_CP;
END_IF   
			
//Read out the cycle time to calculate the energy counters
//Cycle Time in MS
udicycleTime := TwinCAT_SystemInfoVarList._TaskInfo[TaskIndex.index].CycleTime / 10000;

//Calculate the cycles what is needed for 1 Minute
lrCyclesForMinute := UDINT_TO_LREAL((1 * udicycleTime)) / 60000;	

//Calculate past time in hours
lrPastTime := lrPastTime + (lrCyclesForMinute / 60);

//Calculate the Energy when the power data change and start then from new
IF MEMCMP(ADR(lrTotalPower),ADR(lrTotalPower_CP),SIZEOF(lrTotalPower_CP)) <> 0 THEN
	//INFO : Negative Value at the moment is not in use about the limitation of the Total power
	IF lrSumToCalculate < 0 THEN
		lrCounterProduction_CP := lrCounterProduction_CP + (lrSumToCalculate * - 1);
	ELSE
		lrCounterConsumption_CP := lrCounterConsumption_CP + lrSumToCalculate;
	END_IF
		lrSumToCalculate := 0;
			lrPastTime := 0;
				lrTotalPower_CP := lrTotalPower;
END_IF

//Calculate the sum after the calculation why we must calculate after the power change
lrSumToCalculate := lrTotalPower * lrPastTime;

(*-------------------------------------------------------------Service from Backend is ready and check the connection to backen for dissabel/enable Function---------------------------------------------------------------*)

//Try to reset the variable for connection on the GVL. When all is normal then the Lynus Mqtt connection function set this variable to true in the next cycle
//When we have no connection to the backend then after Lynus_Standards.Constants_General.tTimeDissableLynusFunctions days the Function is dissabled with all of his functionalities
timResetConnectionOnGVL(IN:= NOT timResetConnectionOnGVL.Q, PT:= T#1H, Q=> , ET=> );
	IF timResetConnectionOnGVL.Q THEN Lynus_Standards.GVL_Communicator.bStateConnectionToEnableFunctions := FALSE; END_IF
		IF NOT Lynus_Standards.GVL_Communicator.bStateConnectionToEnableFunctions THEN timDissableFunctions.IN := TRUE; ELSE timDissableFunctions.IN := FALSE; END_IF  
			timDissableFunctions(IN:= , PT:= Lynus_Standards.Constants_General.tTimeDissableLynusFunctions, Q=> , ET=> );

(*-----------------------------------------------------------------------------Error ----------------------------------------------------------------------------*)

IF timDissableFunctions.Q THEN fbHouseC.bWarning := TRUE; fbHouseC.iWarningCode := 0; ELSE fbHouseC.bWarning := FALSE; END_IF 	
	IF Lynus_Standards.GVL_Energy.stNumberOfDevices.diNumberOfHouseConsumption > Constants_Energy.diMaxNumberOfHouseConsumptions OR bError THEN fbHouseC.bError := TRUE; ELSE fbHouseC.bError := FALSE; END_IF 
		IF Lynus_Standards.GVL_Energy.stNumberOfDevices.diNumberOfHouseConsumption > Constants_Energy.diMaxNumberOfHouseConsumptions THEN fbHouseC.iErrorCode := 1;
		ELSIF bError THEN fbHouseC.iErrorCode := 0; 
		END_IF  

(*------------------------------------------------------------------FB House----------------------------------------------------------------------------*)	
	
fbHouseC(
	bEnable:= bEnable AND NOT timDissableFunctions.Q,
	bError:= , 
	bWriteWithDelay:= TRUE, 
	iErrorCode:= , 
	iWarningCode:= , 
	lrTotalCounterEnergy_Consumption:= lrCounterConsumption_CP * 1000, 
	lrTotalCounterEnergy_Production:= lrCounterProduction_CP * 1000, 
	lrCounterEnergyT1_Consumption:= lrCounterConsumption_CP * 1000, 
	lrCounterEnergyT2_Consumption:= , 
	lrCounterEnergyT1_Production:= lrCounterProduction_CP * 1000, 
	lrCounterEnergyT2_Production:= , 
	lrPowerHouseConsumption:= lrTotalPower * 1000, 
	tTimDelayOutput:= T#5S, 
	stDataHouseCOut=> , 
	stDataHouseCOutDelay=> stDataHouseC);
	
	(*-----------------------------------------------------------Handle data to Global structure for the House consumption-----------------------------------------------------------------*)

CASE iStateGVLData OF
	
	0://Init Step
		byWaitInStep := 0;
			diCounterForGVL := 1;
	
	1://Wait for 4 Steps before clean al Data on GVL
		byWaitInStep := byWaitInStep + 1;
			IF byWaitInStep >= 4 AND fbNumberDevice.bNumberIsCalculatet THEN iStateGVLData := 2; END_IF
				//To much Devices, back to the Init step
				IF byWaitInStep >= 4 AND NOT fbNumberDevice.bNumberIsCalculatet THEN iStateGVLData := 0; END_IF	
			
	2://Clear all Data in GVL
		Lynus_Standards.GVL_Energy.stDataHouseConsumptions[diCounterForGVL].bEnabled := FALSE;
			Lynus_Standards.GVL_Energy.stDataHouseConsumptions[diCounterForGVL].byErrorWarning := 0;
				Lynus_Standards.GVL_Energy.stDataHouseConsumptions[diCounterForGVL].lrPowerConsumption := 0;
					Lynus_Standards.GVL_Energy.stDataHouseConsumptions[diCounterForGVL].lrPower := 0;
						Lynus_Standards.GVL_Energy.stDataHouseConsumptions[diCounterForGVL].lrPowerProduction := 0;
		
		diCounterForGVL := diCounterForGVL + 1;
			diCounterForGVL := LIMIT(0,diCounterForGVL,Constants_Energy.diMaxNumberOfHouseConsumptions);
				//Back to the init step
				IF diCounterForGVL >= Constants_Energy.diMaxNumberOfHouseConsumptions THEN iStateGVLData := 0; END_IF
				
END_CASE 	 

IF diNrOfHouseC_OUT > 0 AND fbNumberDevice.bNumberIsCalculatet THEN
	Lynus_Standards.GVL_Energy.stDataHouseConsumptions[diNrOfHouseC_OUT].bEnabled := fbHouseC.stDataHouseCOut.bEnabled;
		Lynus_Standards.GVL_Energy.stDataHouseConsumptions[diNrOfHouseC_OUT].byErrorWarning := fbHouseC.stDataHouseCOut.byErrorWarning;
			Lynus_Standards.GVL_Energy.stDataHouseConsumptions[diNrOfHouseC_OUT].lrPowerConsumption := fbHouseC.stDataHouseCOut.lrPowerConsumption;
				Lynus_Standards.GVL_Energy.stDataHouseConsumptions[diNrOfHouseC_OUT].lrPower := fbHouseC.stDataHouseCOut.lrPower;
					Lynus_Standards.GVL_Energy.stDataHouseConsumptions[diNrOfHouseC_OUT].lrPowerProduction := fbHouseC.stDataHouseCOut.lrPowerProduction;
END_IF 	

(*----------------------------------------------------------Save persistent data----------------------------------------------------------------*)

arrPD[1](lrValue:= BOOL_TO_LREAL(bEnable), bEventBasedActive=> );
arrPD[2](lrValue:= DINT_TO_LREAL(diNrOfEMS_IN), bEventBasedActive=> );
arrPD[3](lrValue:= lrCounterConsumption, bEventBasedActive=> );
arrPD[4](lrValue:= lrCounterProduction, bEventBasedActive=> );

END_FUNCTION_BLOCK

// ---- FBs/House Consumption/With Energy Meter/FB_HouseC_Power.TcPOU
{attribute 'hide_all_locals'}
FUNCTION_BLOCK FB_HouseC_Power
VAR_INPUT PERSISTENT
	bEnable									: BOOL;													//{#lynus.ag#()} //Enable the Fuctionblock and his logic
	bPowerDataInvers						: BOOL;													//With True its possible to invert all received power data from the electric meter
	diNrOfEM_IN_HouseC						: DINT;													//Number of the electric meter for incoming power data. (Power Data for this Device)
END_VAR
VAR_INPUT
END_VAR
VAR_OUTPUT
	stDataHouseC							: ST_HouseConsumption_Output;							//{#lynus.ag#()} //House consumption output data
	diNrOfHouseC_OUT						: DINT;													//Active Number from the House connection for using on other functions
END_VAR
VAR
	fbHouseC								: FB_HouseConsumption;									//Function for House consumption
	fbNumberDevice							: FB_NumberOfDevice;									//Function block to calcualte the number of the Device
	timDissableFunctions					: TON;													//Timer to dissable the Function after Lynus_Standards.Constants_General.tTimeDissableLynusFunctions Days without connection to the Lynus Cloud
	timResetConnectionOnGVL					: TON;													//Timer to try reset the connection Flag on the GVL. (When somebody delete the Connection Function and make only a onlinechange)
	arrPD									: ARRAY[1..3] OF FB_PersistentData_Number;				//Function to save persistent data 
	byWaitInStep							: BYTE;													//Wait in Step before start to clean data on PLC
	iStateGVLData							: INT;													//State machine to handle the data on the GVL
	diCounterForGVL							: DINT;													//Counter to clean old data on GVL
END_VAR

//Creator : Kai Ebensperger
//Company : Lynus AG
//Date : 07.06.2021
//Version : 1.0.0.0

//With this function block its possible to show the power data from a house.

//NOTE for diNr.....Designation => 
//_ID = Only Incoming Data to this function
//_OD = Only Outcomming Data from this function
//_IDOD = Incoming Data to this function and outcoming data from this function

(*------------------------------------------------------------Limits----------------------------------------------------------------------------------*)

diNrOfEM_IN_HouseC := LIMIT(0,diNrOfEM_IN_HouseC,Constants_Energy.diMaxNumberOfElectricMeters);	

(*------------------------------------------------------------------Power Data----------------------------------------------------------------------------*)

IF NOT bPowerDataInvers THEN
	fbHouseC.lrCounterEnergyT1_Consumption := Lynus_Standards.GVL_Energy.stDataElectricMeters[diNrOfEM_IN_HouseC].lrCounterEnergyT1_Production * 1000;
	fbHouseC.lrCounterEnergyT2_Consumption := Lynus_Standards.GVL_Energy.stDataElectricMeters[diNrOfEM_IN_HouseC].lrCounterEnergyT2_Production * 1000;
	fbHouseC.lrCounterEnergyT1_Production := Lynus_Standards.GVL_Energy.stDataElectricMeters[diNrOfEM_IN_HouseC].lrCounterEnergyT1_Consumption * 1000;
	fbHouseC.lrCounterEnergyT2_Production := Lynus_Standards.GVL_Energy.stDataElectricMeters[diNrOfEM_IN_HouseC].lrCounterEnergyT1_Consumption * 1000;
	fbHouseC.lrTotalCounterEnergy_Consumption := Lynus_Standards.GVL_Energy.stDataElectricMeters[diNrOfEM_IN_HouseC].lrTotalCounterEnergy_Production * 1000;
	fbHouseC.lrTotalCounterEnergy_Production := Lynus_Standards.GVL_Energy.stDataElectricMeters[diNrOfEM_IN_HouseC].lrTotalCounterEnergy_Consumption * 1000;
		fbHouseC.lrPowerHouseConsumption := (Lynus_Standards.GVL_Energy.stDataElectricMeters[diNrOfEM_IN_HouseC].lrPower * 1000) * - 1;
ELSE
	fbHouseC.lrCounterEnergyT1_Consumption := Lynus_Standards.GVL_Energy.stDataElectricMeters[diNrOfEM_IN_HouseC].lrCounterEnergyT1_Consumption * 1000;
	fbHouseC.lrCounterEnergyT2_Consumption := Lynus_Standards.GVL_Energy.stDataElectricMeters[diNrOfEM_IN_HouseC].lrCounterEnergyT2_Consumption * 1000;
	fbHouseC.lrCounterEnergyT1_Production := Lynus_Standards.GVL_Energy.stDataElectricMeters[diNrOfEM_IN_HouseC].lrCounterEnergyT1_Production * 1000;
	fbHouseC.lrCounterEnergyT2_Production := Lynus_Standards.GVL_Energy.stDataElectricMeters[diNrOfEM_IN_HouseC].lrCounterEnergyT2_Production * 1000;
	fbHouseC.lrTotalCounterEnergy_Consumption := Lynus_Standards.GVL_Energy.stDataElectricMeters[diNrOfEM_IN_HouseC].lrTotalCounterEnergy_Consumption * 1000;
	fbHouseC.lrTotalCounterEnergy_Production := Lynus_Standards.GVL_Energy.stDataElectricMeters[diNrOfEM_IN_HouseC].lrTotalCounterEnergy_Production * 1000;
		fbHouseC.lrPowerHouseConsumption := Lynus_Standards.GVL_Energy.stDataElectricMeters[diNrOfEM_IN_HouseC].lrPower * 1000;
END_IF

(*-------------------------------------------------------------Calcualte the number of House Consumption---------------------------------------------------------------*)

fbNumberDevice(
	diActualNumberOfDevices:= Lynus_Standards.GVL_Energy.stNumberOfDevices.diNumberOfHouseConsumption, 
	diMaxNumberOfDevices:= Constants_Energy.diMaxNumberOfHouseConsumptions, 
	udiCounterOnlineChange:= TwinCAT_SystemInfoVarList._AppInfo.OnlineChangeCnt, 
	bNumberIsCalculatet=> , 
	bFPNumberIsCalculatet=> , 
	bOnlineChange=> , 
	diNumberForThisDevice=> diNrOfHouseC_OUT, 
	diNumberOfTotalDevices=> );

//Write new Numer on GVL
IF fbNumberDevice.bFPNumberIsCalculatet THEN
	Lynus_Standards.GVL_Energy.stNumberOfDevices.diNumberOfHouseConsumption := fbNumberDevice.diNumberOfTotalDevices;	
END_IF 

//Delete old Number on GVL
IF fbNumberDevice.bOnlineChange THEN 
	Lynus_Standards.GVL_Energy.stNumberOfDevices.diNumberOfHouseConsumption := diNrOfHouseC_OUT;	
		iStateGVLData := 1; 
END_IF

(*-------------------------------------------------------------Service from Backend is ready and check the connection to backen for dissabel/enable Function---------------------------------------------------------------*)

//Try to reset the variable for connection on the GVL. When all is normal then the Lynus Mqtt connection function set this variable to true in the next cycle
//When we have no connection to the backend then after Lynus_Standards.Constants_General.tTimeDissableLynusFunctions days the Function is dissabled with all of his functionalities
timResetConnectionOnGVL(IN:= NOT timResetConnectionOnGVL.Q, PT:= T#1H, Q=> , ET=> );
	IF timResetConnectionOnGVL.Q THEN Lynus_Standards.GVL_Communicator.bStateConnectionToEnableFunctions := FALSE; END_IF
		IF NOT Lynus_Standards.GVL_Communicator.bStateConnectionToEnableFunctions THEN timDissableFunctions.IN := TRUE; ELSE timDissableFunctions.IN := FALSE; END_IF  
			timDissableFunctions(IN:= , PT:= Lynus_Standards.Constants_General.tTimeDissableLynusFunctions, Q=> , ET=> );

(*-----------------------------------------------------------------------------Error ----------------------------------------------------------------------------*)

IF timDissableFunctions.Q THEN fbHouseC.bWarning := TRUE; fbHouseC.iWarningCode := 0; ELSE fbHouseC.bWarning := FALSE; END_IF 	
	IF Lynus_Standards.GVL_Energy.stNumberOfDevices.diNumberOfHouseConsumption > Constants_Energy.diMaxNumberOfHouseConsumptions THEN 
		fbHouseC.bError := TRUE; 
			fbHouseC.iErrorCode := 1;
	ELSE 
		fbHouseC.bError := FALSE; 
			fbHouseC.iErrorCode := 0;
	END_IF  
	
(*------------------------------------------------------------------FB House----------------------------------------------------------------------------*)

fbHouseC(
	bEnable:= bEnable AND NOT timDissableFunctions.Q,
	bError:= , 
	bWriteWithDelay:= TRUE, 
	iErrorCode:= , 
	iWarningCode:= , 
	lrTotalCounterEnergy_Consumption:= , 
	lrTotalCounterEnergy_Production:= , 
	lrCounterEnergyT1_Consumption:= , 
	lrCounterEnergyT2_Consumption:= , 
	lrCounterEnergyT1_Production:= , 
	lrCounterEnergyT2_Production:= , 
	lrPowerHouseConsumption:= , 
	tTimDelayOutput:= T#5S, 
	stDataHouseCOut=> , 
	stDataHouseCOutDelay=> stDataHouseC);		
	
(*-----------------------------------------------------------Handle data to Global structure for the House consumption-----------------------------------------------------------------*)

CASE iStateGVLData OF
	
	0://Init Step
		byWaitInStep := 0;
			diCounterForGVL := 1;
	
	1://Wait for 4 Steps before clean al Data on GVL
		byWaitInStep := byWaitInStep + 1;
			IF byWaitInStep >= 4 AND fbNumberDevice.bNumberIsCalculatet THEN iStateGVLData := 2; END_IF
				//To much Devices, back to the Init step
				IF byWaitInStep >= 4 AND NOT fbNumberDevice.bNumberIsCalculatet THEN iStateGVLData := 0; END_IF	
			
	2://Clear all Data in GVL
		Lynus_Standards.GVL_Energy.stDataHouseConsumptions[diCounterForGVL].bEnabled := FALSE;
			Lynus_Standards.GVL_Energy.stDataHouseConsumptions[diCounterForGVL].byErrorWarning := 0;
				Lynus_Standards.GVL_Energy.stDataHouseConsumptions[diCounterForGVL].lrPowerConsumption := 0;
					Lynus_Standards.GVL_Energy.stDataHouseConsumptions[diCounterForGVL].lrPower := 0;
						Lynus_Standards.GVL_Energy.stDataHouseConsumptions[diCounterForGVL].lrPowerProduction := 0;
		
		diCounterForGVL := diCounterForGVL + 1;
			diCounterForGVL := LIMIT(0,diCounterForGVL,Constants_Energy.diMaxNumberOfHouseConsumptions);
				//Back to the init step
				IF diCounterForGVL >= Constants_Energy.diMaxNumberOfHouseConsumptions THEN iStateGVLData := 0; END_IF

END_CASE 	 

IF diNrOfHouseC_OUT > 0 AND fbNumberDevice.bNumberIsCalculatet THEN
	Lynus_Standards.GVL_Energy.stDataHouseConsumptions[diNrOfHouseC_OUT].bEnabled := fbHouseC.stDataHouseCOut.bEnabled;
		Lynus_Standards.GVL_Energy.stDataHouseConsumptions[diNrOfHouseC_OUT].byErrorWarning := fbHouseC.stDataHouseCOut.byErrorWarning;
			Lynus_Standards.GVL_Energy.stDataHouseConsumptions[diNrOfHouseC_OUT].lrPowerConsumption := fbHouseC.stDataHouseCOut.lrPowerConsumption;
				Lynus_Standards.GVL_Energy.stDataHouseConsumptions[diNrOfHouseC_OUT].lrPower := fbHouseC.stDataHouseCOut.lrPower;
					Lynus_Standards.GVL_Energy.stDataHouseConsumptions[diNrOfHouseC_OUT].lrPowerProduction := fbHouseC.stDataHouseCOut.lrPowerProduction;
END_IF 	

(*----------------------------------------------------------Save persistent data----------------------------------------------------------------*)

arrPD[1](lrValue:= BOOL_TO_LREAL(bEnable), bEventBasedActive=> );
arrPD[2](lrValue:= BOOL_TO_LREAL(bPowerDataInvers), bEventBasedActive=> );
arrPD[3](lrValue:= DINT_TO_LREAL(diNrOfEM_IN_HouseC), bEventBasedActive=> );

END_FUNCTION_BLOCK

// ---- FBs/KNX Master/FB_KL6301_KNX_Master.TcPOU
FUNCTION_BLOCK FB_KL6301_KNX_Master
VAR_INPUT PERSISTENT
	stPhysAddrTerminal						: EIB_PHYS_ADDR;								//Physical KNX Adress for the KL6301 Terminal. Must be unique throughout the KNX network.
	arrGroupFilter							: ARRAY[1..8] OF EIB_GROUP_FILTER;				//Group Filter. Here all group addresses per group must be entered which may pass the filter to KL6301. All other group addresses are ignored.
	iKL6301Mode								: INT;											//Work Mode from the KL6301. 0 = 4 Filters with 64 Entrys with FW B0 or higher. 1 = 8 Filters with 32 Entrys with FW B1 or higher. 2 = 8 Filters with 32 Entrys with FW B3 or higher. 100 = Only Monitoring function with FW B1 or higher.	
END_VAR
VAR_INPUT
	uiKBusState_IN							: UINT;											//K-Bus State from the K-Bus Box on wich the Terminal is connected. (Connect with FB_K_Bus_state)
END_VAR
VAR_OUTPUT
	bActive									: BOOL;											//Function is Active
	bReady									: BOOL;											//Function is Ready
	byErrorWarning							: BYTE;											//Error Warning State
	diNrOfKNXMasterLine_OUT					: DINT;											//Active Number from the KNX Master Function for using on other functions
	eMessageKNXMaster						: E_Message_KNXMaster;							//Message from the KNX Master Function
END_VAR
VAR
	{attribute 'hide'}
	fbKNXMaster								: KL6301;										//KNX Master for KL6301
	{attribute 'hide'}
	fbNumberDevice							: FB_NumberOfDevice;							//Function block to calcualte the number of the Device
	{attribute 'hide'}
	fbKNXMessage							: FB_KNXMaster_Messages;						//KNX Messages
	{attribute 'hide'}
	arrPD									: ARRAY[1..36] OF FB_PersistentData_Number;		//FB Persistent Data
	{attribute 'hide'}
	timDissableFunctions					: TON;											//Timer to dissable the Function after Lynus_Standards.Constants_General.tTimeDissableLynusFunctions Days without connection to the Lynus Cloud
	{attribute 'hide'}
	timResetConnectionOnGVL					: TON;											//Timer to try reset the connection Flag on the GVL. (When somebody delete the Connection Function and make only a onlinechange)
	{attribute 'hide'}
	timActive								: TON;											//Timer to activate the Terminal
	{attribute 'hide'}
	fbGetTask								: GETCURTASKINDEX;								//Task Index
	arrKNXKL6301ComIn        	AT%I*	 	: ARRAY[1..24] OF BYTE;							//Input Array for the KL6301 to map on the KL6301 Terminal
	arrKNXKL6301ComOut        	AT%Q*		: ARRAY[1..24] OF BYTE;							//Output Array for the KL6301 to map on the KL6301 Terminal
	{attribute 'hide'}
	stDefaultKNXCom							: EIB_REC;										//Default structure to set the GVL for the KNX communication to default values
	{attribute 'hide'}
	bActivateKL6301							: BOOL;											//Activate the KL6301
	{attribute 'hide'}
	byWaitInStep							: BYTE;											//Wait in Step before start to clean data on PLC
	{attribute 'hide'}
	byLPLimitFilter							: BYTE;											//Loop to ckeck the Limits for the KNX Filters
	{attribute 'hide'}
	iStateGVLData							: INT;											//State machine to handle the data on the GVL
	{attribute 'hide'}
	diCounterForGVL							: DINT;											//Counter to clean old data on GVL
END_VAR

//Creator : Kai Ebensperger
//Company : Lynus AG
//Date : 24.07.2021
//Version : 1.0.0.0

//With this function block we can communicate with a beckhoff KL6301 KNX Terminal.
//This Functionblock receive and send the data to the KNX Bus from ther other KNX Read and Write functions in the plc.
//This Functions block must insert in the same task with all other knx functions from the plc
//In the PLC project this block may only be called once per cycle!
//A PLC project may contain a maximum of 64 KL6301! We limit by ourself in the constants
//On the Inputs the user must set the physical KNX Adress for the Terminal. Must be unique throughout the KNX network.
//In addition, all group addresses that must pass through to the terminal must be entered in the group filters. Depending on the mode of the terminal, you can specify between 4 and 8 groupfilters with 32 or 64 entries each.
//iMode:
//0 - For firmware B0 and higher - 4 filters a 64 entries
//1 - For firmware B1 and higher - 8 filters a 32 entries
//2 - For firmware B3 and higher - 8 filters a 32 entries inverted. For cross communication of telegrams within the EIB/KNX network, which are not connected to the KL6301, it must be ensured that these group addresses are included in the filter, so that the terminal does not send an ACK.
//100 - For firmware B1 and higher - Monitor function, all group address telegrams are received. The telegrams are not acknowledged (no ACK is sent). In monitor mode, it is not possible to send.

//NOTE for diNr.....Designation => 
//_IN = Here Data come in from other Functions or go out to other functions about the GVL
//_OUT = Here Data go out to other functions about the GVL

(*------------------------------------------------------------Limits----------------------------------------------------------------------------------*)

stPhysAddrTerminal.Area := LIMIT(0,stPhysAddrTerminal.Area,15);
	stPhysAddrTerminal.Line := LIMIT(0,stPhysAddrTerminal.Line,15);	
		iKL6301Mode := LIMIT(0,iKL6301Mode,100);
		
//Group Filters
FOR byLPLimitFilter := 1 TO 8 BY 1 DO
	arrGroupFilter[byLPLimitFilter].GROUP_LEN := LIMIT(0,arrGroupFilter[byLPLimitFilter].GROUP_LEN,63);
	arrGroupFilter[byLPLimitFilter].GROUP_ADDR.MAIN := LIMIT(0,arrGroupFilter[byLPLimitFilter].GROUP_ADDR.MAIN,31);
	arrGroupFilter[byLPLimitFilter].GROUP_ADDR.SUB_MAIN := LIMIT(0,arrGroupFilter[byLPLimitFilter].GROUP_ADDR.SUB_MAIN,7);
END_FOR
	
(*-------------------------------------------------------------Calcualte the number of KNX Master---------------------------------------------------------------*)

fbNumberDevice(
	diActualNumberOfDevices:= Lynus_Standards.GVL_Bussystems.diNumberOfKNXMasters, 
	diMaxNumberOfDevices:= Constants_Bussystems.diMaxNumberOfKNXMasterKL6301, 
	udiCounterOnlineChange:= TwinCAT_SystemInfoVarList._AppInfo.OnlineChangeCnt, 
	bNumberIsCalculatet=> , 
	bFPNumberIsCalculatet=> , 
	bOnlineChange=> , 
	diNumberForThisDevice=> diNrOfKNXMasterLine_OUT, 
	diNumberOfTotalDevices=> );

//Write new Numer on GVL
IF fbNumberDevice.bFPNumberIsCalculatet THEN
	Lynus_Standards.GVL_Bussystems.diNumberOfKNXMasters := fbNumberDevice.diNumberOfTotalDevices;	
END_IF 

//Delete old Number on GVL
IF fbNumberDevice.bOnlineChange THEN 
	Lynus_Standards.GVL_Bussystems.diNumberOfKNXMasters := diNrOfKNXMasterLine_OUT;	
		iStateGVLData := 1; 
END_IF	

(*-------------------------------------------------------------Service from Backend is ready and check the connection to backen for dissabel/enable Function---------------------------------------------------------------*)

//Try to reset the variable for connection on the GVL. When all is normal then the Lynus Mqtt connection function set this variable to true in the next cycle
//When we have no connection to the backend then after Lynus_Standards.Constants_General.tTimeDissableLynusFunctions days the Function is dissabled with all of his functionalities
timResetConnectionOnGVL(IN:= NOT timResetConnectionOnGVL.Q, PT:= T#1H, Q=> , ET=> );
	IF timResetConnectionOnGVL.Q THEN Lynus_Standards.GVL_Communicator.bStateConnectionToEnableFunctions := FALSE; END_IF
		IF NOT Lynus_Standards.GVL_Communicator.bStateConnectionToEnableFunctions THEN timDissableFunctions.IN := TRUE; ELSE timDissableFunctions.IN := FALSE; END_IF  
			timDissableFunctions(IN:= , PT:= Lynus_Standards.Constants_General.tTimeDissableLynusFunctions, Q=> , ET=> );
			
(*-------------------------------------------------------------KNX Master---------------------------------------------------------------*)

//Activate the Terminal
timActive(IN:= uiKBusState_IN = 0, PT:= T#500MS, Q=> , ET=> );
	IF timActive.Q THEN bActivateKL6301 := TRUE; END_IF 

fbGetTask(index=> );	
	IF TwinCAT_SystemInfoVarList._TaskInfo[fbGetTask.index].FirstCycle THEN bActivateKL6301 := FALSE; END_IF	
	
IF NOT timDissableFunctions.Q AND diNrOfKNXMasterLine_OUT <> 0 AND fbNumberDevice.bNumberIsCalculatet AND bActivateKL6301 THEN fbKNXMaster.bActivate := TRUE; END_IF
	IF timDissableFunctions.Q OR diNrOfKNXMasterLine_OUT <= 0 OR NOT fbNumberDevice.bNumberIsCalculatet OR NOT bActivateKL6301 THEN fbKNXMaster.bActivate := FALSE; END_IF

fbKNXMaster(
	bActivate:= , 
	idx:= DINT_TO_INT(diNrOfKNXMasterLine_OUT), 
	EIB_PHYS_ADDR:= stPhysAddrTerminal, 
	EIB_GROUP_FILTER:= arrGroupFilter, 
	iMode:= iKL6301Mode, 
	tTimeout:= T#5S, 
	bActive=> bActive, 
	bReady=> bReady, 
	bError=> , 
	iErrorId=> , 
	str_Data_Rec=> Lynus_Standards.GVL_Bussystems.stDataOfKNXMasterKL6301[diNrOfKNXMasterLine_OUT], 
	KL6301_IN:= arrKNXKL6301ComIn, 
	KL6301_OUT:= arrKNXKL6301ComOut);

(*------------------------------------------------------------------Error and Warning----------------------------------------------------------------------------*)
			
IF timDissableFunctions.Q THEN fbKNXMessage.bWarning := TRUE; fbKNXMessage.iWarningCode := 0; ELSE fbKNXMessage.bWarning := FALSE; END_IF   
	IF (Lynus_Standards.GVL_Bussystems.diNumberOfKNXMasters > Constants_Bussystems.diMaxNumberOfKNXMasterKL6301) THEN 
		fbKNXMessage.bErrorIntern := TRUE;
			fbKNXMessage.iErrorCode := 1;
	ELSE
		fbKNXMessage.bErrorIntern := FALSE;
	END_IF	

IF fbKNXMaster.bError THEN 
	fbKNXMessage.bErrorKNX := TRUE;
		fbKNXMessage.iErrorCode := fbKNXMaster.iErrorId;
ELSE
	IF NOT fbKNXMaster.bError THEN 
		fbKNXMessage.bErrorKNX := FALSE;
	END_IF
END_IF	
		
fbKNXMessage(
	bErrorKNX:= , 
	bErrorIntern:= , 
	bWarning:= , 
	iWarningCode:= , 
	iErrorCode:= , 
	byErrorWarning=> byErrorWarning, 
	eMessageKNXMaster=> eMessageKNXMaster);
	
(*-----------------------------------------------------------Handle data to Global structure for KNX Communication-----------------------------------------------------------------*)
	
CASE iStateGVLData OF
	
	0://Init Step
		byWaitInStep := 0;
			diCounterForGVL := 1;
	
	1://Wait for 4 Steps before clean al Data on GVL
		byWaitInStep := byWaitInStep + 1;
			IF byWaitInStep >= 4 AND fbNumberDevice.bNumberIsCalculatet THEN iStateGVLData := 2; END_IF
				//To much Devices, back to the Init step
				IF byWaitInStep >= 4 AND NOT fbNumberDevice.bNumberIsCalculatet THEN iStateGVLData := 0; END_IF	
			
	2://Clear all Data in GVL
	//Some Parts in the GVL Reset the Slave. Otherwise there will be problems when writing the new addresses to the array in the GVL.
	
	Lynus_Standards.GVL_Bussystems.stDataOfKNXMasterKL6301[diCounterForGVL] := stDefaultKNXCom;
														 		
		diCounterForGVL := diCounterForGVL + 1;
			diCounterForGVL := LIMIT(0,diCounterForGVL,Constants_Bussystems.diMaxNumberOfKNXMasterKL6301);
				//Back to the init step
				IF diCounterForGVL >= Constants_Bussystems.diMaxNumberOfKNXMasterKL6301 THEN iStateGVLData := 0; END_IF

END_CASE 

(*----------------------------------------------------------Save persistent data----------------------------------------------------------------*)

arrPD[1](lrValue:= BYTE_TO_LREAL(stPhysAddrTerminal.Area), bEventBasedActive=> );
arrPD[2](lrValue:= BYTE_TO_LREAL(stPhysAddrTerminal.Device), bEventBasedActive=> );
arrPD[3](lrValue:= BYTE_TO_LREAL(stPhysAddrTerminal.Line), bEventBasedActive=> );
arrPD[4](lrValue:= BYTE_TO_LREAL(arrGroupFilter[1].GROUP_ADDR.MAIN), bEventBasedActive=> );
arrPD[5](lrValue:= BYTE_TO_LREAL(arrGroupFilter[1].GROUP_ADDR.NUMBER), bEventBasedActive=> );
arrPD[6](lrValue:= BYTE_TO_LREAL(arrGroupFilter[1].GROUP_ADDR.SUB_MAIN), bEventBasedActive=> );
arrPD[7](lrValue:= WORD_TO_LREAL(arrGroupFilter[1].GROUP_LEN), bEventBasedActive=> );
arrPD[8](lrValue:= BYTE_TO_LREAL(arrGroupFilter[2].GROUP_ADDR.MAIN), bEventBasedActive=> );
arrPD[9](lrValue:= BYTE_TO_LREAL(arrGroupFilter[2].GROUP_ADDR.NUMBER), bEventBasedActive=> );
arrPD[10](lrValue:= BYTE_TO_LREAL(arrGroupFilter[2].GROUP_ADDR.SUB_MAIN), bEventBasedActive=> );
arrPD[11](lrValue:= WORD_TO_LREAL(arrGroupFilter[2].GROUP_LEN), bEventBasedActive=> );
arrPD[12](lrValue:= BYTE_TO_LREAL(arrGroupFilter[3].GROUP_ADDR.MAIN), bEventBasedActive=> );
arrPD[13](lrValue:= BYTE_TO_LREAL(arrGroupFilter[3].GROUP_ADDR.NUMBER), bEventBasedActive=> );
arrPD[14](lrValue:= BYTE_TO_LREAL(arrGroupFilter[3].GROUP_ADDR.SUB_MAIN), bEventBasedActive=> );
arrPD[15](lrValue:= WORD_TO_LREAL(arrGroupFilter[3].GROUP_LEN), bEventBasedActive=> );
arrPD[16](lrValue:= BYTE_TO_LREAL(arrGroupFilter[4].GROUP_ADDR.MAIN), bEventBasedActive=> );
arrPD[17](lrValue:= BYTE_TO_LREAL(arrGroupFilter[4].GROUP_ADDR.NUMBER), bEventBasedActive=> );
arrPD[18](lrValue:= BYTE_TO_LREAL(arrGroupFilter[4].GROUP_ADDR.SUB_MAIN), bEventBasedActive=> );
arrPD[19](lrValue:= WORD_TO_LREAL(arrGroupFilter[4].GROUP_LEN), bEventBasedActive=> );
arrPD[20](lrValue:= BYTE_TO_LREAL(arrGroupFilter[5].GROUP_ADDR.MAIN), bEventBasedActive=> );
arrPD[21](lrValue:= BYTE_TO_LREAL(arrGroupFilter[5].GROUP_ADDR.NUMBER), bEventBasedActive=> );
arrPD[22](lrValue:= BYTE_TO_LREAL(arrGroupFilter[5].GROUP_ADDR.SUB_MAIN), bEventBasedActive=> );
arrPD[23](lrValue:= WORD_TO_LREAL(arrGroupFilter[5].GROUP_LEN), bEventBasedActive=> );
arrPD[24](lrValue:= BYTE_TO_LREAL(arrGroupFilter[6].GROUP_ADDR.MAIN), bEventBasedActive=> );
arrPD[25](lrValue:= BYTE_TO_LREAL(arrGroupFilter[6].GROUP_ADDR.NUMBER), bEventBasedActive=> );
arrPD[26](lrValue:= BYTE_TO_LREAL(arrGroupFilter[6].GROUP_ADDR.SUB_MAIN), bEventBasedActive=> );
arrPD[27](lrValue:= WORD_TO_LREAL(arrGroupFilter[6].GROUP_LEN), bEventBasedActive=> );
arrPD[28](lrValue:= BYTE_TO_LREAL(arrGroupFilter[7].GROUP_ADDR.MAIN), bEventBasedActive=> );
arrPD[29](lrValue:= BYTE_TO_LREAL(arrGroupFilter[7].GROUP_ADDR.NUMBER), bEventBasedActive=> );
arrPD[30](lrValue:= BYTE_TO_LREAL(arrGroupFilter[7].GROUP_ADDR.SUB_MAIN), bEventBasedActive=> );
arrPD[31](lrValue:= WORD_TO_LREAL(arrGroupFilter[7].GROUP_LEN), bEventBasedActive=> );
arrPD[32](lrValue:= BYTE_TO_LREAL(arrGroupFilter[8].GROUP_ADDR.MAIN), bEventBasedActive=> );
arrPD[33](lrValue:= BYTE_TO_LREAL(arrGroupFilter[8].GROUP_ADDR.NUMBER), bEventBasedActive=> );
arrPD[34](lrValue:= BYTE_TO_LREAL(arrGroupFilter[8].GROUP_ADDR.SUB_MAIN), bEventBasedActive=> );
arrPD[35](lrValue:= WORD_TO_LREAL(arrGroupFilter[8].GROUP_LEN), bEventBasedActive=> );
arrPD[36](lrValue:= INT_TO_LREAL(iKL6301Mode), bEventBasedActive=> );

END_FUNCTION_BLOCK

// ---- FBs/Meter/Extern/FB_EM_Electric_3P_Ext_Input.TcPOU
FUNCTION_BLOCK FB_EM_Electric_3P_Ext_Input
VAR_INPUT PERSISTENT
	bEnable									: BOOL;											//Enable the function
	bPowerDataInvers						: BOOL;											//power Data Invers
END_VAR
VAR_INPUT
	bErrorExt								: BOOL;											//Error from external Function
	bWarningExt								: BOOL;											//Warning from external Function
	lrTotalCounterEnergy_Consumption		: LREAL;										//Total Counter for Energy consumption with unit kWh
	lrTotalCounterEnergy_Production			: LREAL;										//Total Counter for Energy production with unit kWh
	lrCounterEnergyT1_Consumption			: LREAL;										//Total counter for energy Tariff 1 consumption with unit kWh
	lrCounterEnergyT2_Consumption			: LREAL;										//Total counter for energy Tariff 2 consumption with unit kWh
	lrCounterEnergyT1_Production			: LREAL;										//Total counter for energy Tariff 1 production with unit kWh
	lrCounterEnergyT2_Production			: LREAL;										//Total counter for energy Tariff 2 production with unit kWh
	lrCurrentL1								: LREAL;										//Current from L1 with unit A
	lrVoltageL1N							: LREAL;										//Voltage L1-N with unit V
	lrVoltageL1L2							: LREAL;										//Voltage L1-L2 with unit V
	lrPowerL1								: LREAL;										//Power L1 with unit W
	lrCurrentL2								: LREAL;										//Current from L2 with unit A
	lrVoltageL2N							: LREAL;										//Voltage L2-N with unit V
	lrVoltageL2L3							: LREAL;										//Voltage L2-L3 with unit V
	lrPowerL2								: LREAL;										//Power L2 with unit W
	lrCurrentL3								: LREAL;										//Current from L3 with unit A
	lrVoltageL3N							: LREAL;										//Voltage L3-N with unit V
	lrVoltageL3L1							: LREAL;										//Voltage L3-L1 with unit V
	lrPowerL3								: LREAL;										//Power L3 with unit W
	lrPowerTotal							: LREAL;										//Total power with unit W	
	lrFrequency								: LREAL;										//Frequency with unit HZ
	lrReactivePowerTotal					: LREAL;										//Reactive power with unit var
	lrApparentPowerTotal					: LREAL;										//Apparent Power with unit VA
END_VAR
VAR_OUTPUT
	stDataEMPower							: ST_ElectricMeter_Output_Power;				//Output structure with Data from Electric Meter (Power Data)
	stDataEMCounter							: ST_ElectricMeter_Output_Counter;				//Output structure with Data from Electric Meter (Counter Data)
	diNrOfEM_OUT							: DINT;											//Active Number from the Electric Meter for using on other functions
END_VAR
VAR
	{attribute 'conditionalshow'}
	fbEM									: FB_ElectricMeter;								//Electric Meter Function
	{attribute 'hide'}
	fbNumberDevice							: FB_NumberOfDevice;							//Function block to calcualte the number of the Device
	{attribute 'hide'}
	timDissableFunctions					: TON;											//Timer to dissable the Function after Lynus_Standards.Constants_General.tTimeDissableLynusFunctions Days without connection to the Lynus Cloud
	{attribute 'hide'}
	timResetConnectionOnGVL					: TON;											//Timer to try reset the connection Flag on the GVL. (When somebody delete the Connection Function and make only a onlinechange)
	{attribute 'hide'}
	fbPD									: FB_PersistentData_Number;						//Function to save persistent data
	{attribute 'hide'}
	byWaitInStep							: BYTE;											//Wait in Step before start to clean data on PLC
	{attribute 'hide'}
	iStateGVLData							: INT;											//State machine to handle the data on the GVL
	{attribute 'hide'}
	diCounterForGVL							: DINT;											//Counter to clean old data on GVL
	{attribute 'hide'}
	lrTotalCounterEnergy_Consumption_CP		: LREAL;										//Total Counter for Energy consumption with unit kWh
	{attribute 'hide'}
	lrTotalCounterEnergy_Production_CP		: LREAL;										//Total Counter for Energy production with unit kWh
	{attribute 'hide'}
	lrCounterEnergyT1_Consumption_CP		: LREAL;										//Total counter for energy Tariff 1 consumption with unit kWh
	{attribute 'hide'}
	lrCounterEnergyT2_Consumption_CP		: LREAL;										//Total counter for energy Tariff 2 consumption with unit kWh
	{attribute 'hide'}
	lrCounterEnergyT1_Production_CP			: LREAL;										//Total counter for energy Tariff 1 production with unit kWh
	{attribute 'hide'}
	lrCounterEnergyT2_Production_CP			: LREAL;										//Total counter for energy Tariff 2 production with unit kWh
END_VAR

//Creator : Kai Ebensperger
//Company : Lynus AG
//Date : 05.11.2021
//Version : 1.0.0.0

//With this function block its possible to read in external data from a Electric meter
//This Function is Helpfull when we receive Energy Data from a External Function and we want to write on th GVL from the Electric meter.
//So we can deliver the Energy data on all other Functions in Lynus (Heating Pumps, Electric heating Elemt, ECS, Big consumer....)

//NOTE for diNr.....Designation => 
//_IN = Here Data come in from other Functions or go out to other functions about the GVL
//_OUT = Here Data go out to other functions about the GVL

(*-------------------------------------------------------------Calcualte the number of EM---------------------------------------------------------------*)

fbNumberDevice(
	diActualNumberOfDevices:= Lynus_Standards.GVL_Energy.stNumberOfDevices.diNumberOfElectricMeters, 
	diMaxNumberOfDevices:= Constants_Energy.diMaxNumberOfElectricMeters, 
	udiCounterOnlineChange:= TwinCAT_SystemInfoVarList._AppInfo.OnlineChangeCnt, 
	bNumberIsCalculatet=> , 
	bFPNumberIsCalculatet=> , 
	bOnlineChange=> , 
	diNumberForThisDevice=> diNrOfEM_OUT, 
	diNumberOfTotalDevices=> );

//Write new Numer on GVL
IF fbNumberDevice.bFPNumberIsCalculatet THEN
	Lynus_Standards.GVL_Energy.stNumberOfDevices.diNumberOfElectricMeters := fbNumberDevice.diNumberOfTotalDevices;	
END_IF

//Delete old Number on GVL
IF fbNumberDevice.bOnlineChange THEN 
	Lynus_Standards.GVL_Energy.stNumberOfDevices.diNumberOfElectricMeters := diNrOfEM_OUT;	
		iStateGVLData := 1; 
END_IF

(*-------------------------------------------------------------Service from Backend is ready and check the connection to backen for dissabel/enable Function---------------------------------------------------------------*)

//Try to reset the variable for connection on the GVL. When all is normal then the Lynus Mqtt connection function set this variable to true in the next cycle
//When we have no connection to the backend then after Lynus_Standards.Constants_General.tTimeDissableLynusFunctions days the Function is dissabled with all of his functionalities
timResetConnectionOnGVL(IN:= NOT timResetConnectionOnGVL.Q, PT:= T#1H, Q=> , ET=> );
	IF timResetConnectionOnGVL.Q THEN Lynus_Standards.GVL_Communicator.bStateConnectionToEnableFunctions := FALSE; END_IF
		IF NOT Lynus_Standards.GVL_Communicator.bStateConnectionToEnableFunctions THEN timDissableFunctions.IN := TRUE; ELSE timDissableFunctions.IN := FALSE; END_IF  
			timDissableFunctions(IN:= , PT:= Lynus_Standards.Constants_General.tTimeDissableLynusFunctions, Q=> , ET=> );

(*----------------------------------------------------------------------------------------Electric Meter Function for Pv----------------------------------------------------------------------------------------------*)


//Error and Warning
IF timDissableFunctions.Q OR bWarningExt THEN fbEM.bWarning := TRUE;
ELSE fbEM.bWarning := FALSE; END_IF 
	IF Lynus_Standards.GVL_Energy.stNumberOfDevices.diNumberOfElectricMeters > Constants_Energy.diMaxNumberOfElectricMeters OR bErrorExt THEN fbEM.bError := TRUE; ELSE fbEM.bError := FALSE; END_IF
		IF Lynus_Standards.GVL_Energy.stNumberOfDevices.diNumberOfElectricMeters > Constants_Energy.diMaxNumberOfElectricMeters THEN fbEM.iErrorCode := 1;
		ELSIF bErrorExt THEN fbEM.iErrorCode := 0;
		END_IF

IF timDissableFunctions.Q THEN fbEM.iWarningCode := 0;
ELSIF bWarningExt THEN fbEM.iWarningCode := 1;
END_IF  		
	
//Write the counter values after a change on the inputs
fbEM.bReadOutDataDone := FALSE;
	IF lrTotalCounterEnergy_Consumption <> lrTotalCounterEnergy_Consumption_CP OR lrTotalCounterEnergy_Production <> lrTotalCounterEnergy_Production_CP OR lrCounterEnergyT1_Consumption <> lrCounterEnergyT1_Consumption_CP OR
		lrCounterEnergyT2_Consumption <> lrCounterEnergyT2_Consumption_CP OR lrCounterEnergyT1_Production <> lrCounterEnergyT1_Production_CP OR lrCounterEnergyT2_Production <> lrCounterEnergyT2_Production_CP THEN
			fbEM.bReadOutDataDone := TRUE;
				lrTotalCounterEnergy_Consumption_CP := lrTotalCounterEnergy_Consumption;
					lrTotalCounterEnergy_Production_CP := lrTotalCounterEnergy_Production;
						lrCounterEnergyT1_Consumption_CP := lrCounterEnergyT1_Consumption;
							lrCounterEnergyT2_Consumption_CP := lrCounterEnergyT2_Consumption;
								lrCounterEnergyT1_Production_CP := lrCounterEnergyT1_Production;
									lrCounterEnergyT2_Production_CP := lrCounterEnergyT2_Production;
	END_IF		
		
//Function
fbEM(
	bEnable:= bEnable AND NOT timDissableFunctions.Q, 
	bError:= , 
	bEnableReadOutFunction:= FALSE, 
	bWriteWithDelay:= TRUE, 
	bPowerDataInvers:= bPowerDataInvers,
	bReadOutDataDone:= ,
	iTimeReadOutInterval:= 0, 
	iErrorCode:= , 
	iWarningCode:= , 
	lrTotalCounterEnergy_Consumption:= lrTotalCounterEnergy_Consumption, 
	lrTotalCounterEnergy_Production:= lrTotalCounterEnergy_Production, 
	lrCounterEnergyT1_Consumption:= lrCounterEnergyT1_Consumption, 
	lrCounterEnergyT2_Consumption:= lrCounterEnergyT2_Consumption, 
	lrCounterEnergyT1_Production:= lrCounterEnergyT1_Production, 
	lrCounterEnergyT2_Production:= lrCounterEnergyT2_Production, 
	lrCurrentL1:= lrCurrentL1, 
	lrVoltageL1N:= lrVoltageL1N, 
	lrVoltageL1L2:= lrVoltageL1L2, 
	lrPowerL1:= lrPowerL1, 
	lrCurrentL2:= lrCurrentL2, 
	lrVoltageL2N:= lrVoltageL2N, 
	lrVoltageL2L3:= lrVoltageL2L3, 
	lrPowerL2:= lrPowerL2, 
	lrCurrentL3:= lrCurrentL3, 
	lrVoltageL3N:= lrVoltageL3N, 
	lrVoltageL3L1:= lrVoltageL3L1, 
	lrPowerL3:= lrPowerL3, 
	lrPowerTotal:= lrPowerTotal, 
	lrFrequency:= lrFrequency, 
	lrReactivePowerTotal:= lrReactivePowerTotal, 
	lrApparentPowerTotal:= lrApparentPowerTotal, 
	tTimDelayOutput:= T#5S, 
	stDataEMOutPower=> , 
	stDataEMOutPowerDelay=> stDataEMPower, 
	stDataEMOutCounter=> ,
	stDataEMOutCounterDelay=> stDataEMCounter,
	bReadOutMeter=> );
	
(*-----------------------------------------------------------Handle data to Global structure for Electric Meter-----------------------------------------------------------------*)

CASE iStateGVLData OF
	
	0://Init Step
		byWaitInStep := 0;
			diCounterForGVL := 1;
	
	1://Wait for 4 Steps before clean al Data on GVL
		byWaitInStep := byWaitInStep + 1;
			IF byWaitInStep >= 4 AND fbNumberDevice.bNumberIsCalculatet THEN iStateGVLData := 2; END_IF
				//To much Devices, back to the Init step
				IF byWaitInStep >= 4 AND NOT fbNumberDevice.bNumberIsCalculatet THEN iStateGVLData := 0; END_IF	
			
	2://Clear all Data in GVL
		Lynus_Standards.GVL_Energy.stDataElectricMeters[diCounterForGVL].bEnabled := FALSE;	
			Lynus_Standards.GVL_Energy.stDataElectricMeters[diCounterForGVL].byErrorWarning := 0;
				Lynus_Standards.GVL_Energy.stDataElectricMeters[diCounterForGVL].lrCounterEnergyT1_Consumption := 0;
					Lynus_Standards.GVL_Energy.stDataElectricMeters[diCounterForGVL].lrCounterEnergyT1_Production := 0;
						Lynus_Standards.GVL_Energy.stDataElectricMeters[diCounterForGVL].lrCounterEnergyT2_Consumption := 0;
							Lynus_Standards.GVL_Energy.stDataElectricMeters[diCounterForGVL].lrCounterEnergyT2_Production := 0;
								Lynus_Standards.GVL_Energy.stDataElectricMeters[diCounterForGVL].lrPower := 0;
									Lynus_Standards.GVL_Energy.stDataElectricMeters[diCounterForGVL].lrPowerConsumption := 0;
										Lynus_Standards.GVL_Energy.stDataElectricMeters[diCounterForGVL].lrPowerProduction := 0;
											Lynus_Standards.GVL_Energy.stDataElectricMeters[diCounterForGVL].lrTotalCounterEnergy_Consumption := 0;
												Lynus_Standards.GVL_Energy.stDataElectricMeters[diCounterForGVL].lrTotalCounterEnergy_Production := 0;
		
		//Electric Meters
		diCounterForGVL := diCounterForGVL + 1;
			diCounterForGVL := LIMIT(0,diCounterForGVL,Constants_Energy.diMaxNumberOfElectricMeters);
				//Back to the init step
				IF diCounterForGVL >= Constants_Energy.diMaxNumberOfElectricMeters THEN iStateGVLData := 0; END_IF

END_CASE 	 

//Write Data on GVL for Electric Meter
IF diNrOfEM_OUT > 0 AND fbNumberDevice.bNumberIsCalculatet THEN
	Lynus_Standards.GVL_Energy.stDataElectricMeters[diNrOfEM_OUT].bEnabled := fbEM.stDataEMOutPower.bEnabled;
		Lynus_Standards.GVL_Energy.stDataElectricMeters[diNrOfEM_OUT].byErrorWarning := fbEM.stDataEMOutPower.byErrorWarning;
			Lynus_Standards.GVL_Energy.stDataElectricMeters[diNrOfEM_OUT].lrCounterEnergyT1_Consumption := fbEM.stDataEMOutCounter.lrCounterEnergyT1_Consumption;
				Lynus_Standards.GVL_Energy.stDataElectricMeters[diNrOfEM_OUT].lrCounterEnergyT1_Production := fbEM.stDataEMOutCounter.lrCounterEnergyT1_Production;
					Lynus_Standards.GVL_Energy.stDataElectricMeters[diNrOfEM_OUT].lrCounterEnergyT2_Consumption := fbEM.stDataEMOutCounter.lrCounterEnergyT2_Consumption;
						Lynus_Standards.GVL_Energy.stDataElectricMeters[diNrOfEM_OUT].lrCounterEnergyT2_Production := fbEM.stDataEMOutCounter.lrCounterEnergyT2_Production;		
							Lynus_Standards.GVL_Energy.stDataElectricMeters[diNrOfEM_OUT].lrPower := fbEM.stDataEMOutPower.lrPowerTotal;
								Lynus_Standards.GVL_Energy.stDataElectricMeters[diNrOfEM_OUT].lrPowerConsumption := fbEM.stDataEMOutPower.lrPowerConsumption;
									Lynus_Standards.GVL_Energy.stDataElectricMeters[diNrOfEM_OUT].lrPowerProduction := fbEM.stDataEMOutPower.lrPowerProduction;
										Lynus_Standards.GVL_Energy.stDataElectricMeters[diNrOfEM_OUT].lrTotalCounterEnergy_Consumption := fbEM.stDataEMOutCounter.lrTotalCounterEnergy_Consumption;
											Lynus_Standards.GVL_Energy.stDataElectricMeters[diNrOfEM_OUT].lrTotalCounterEnergy_Production := fbEM.stDataEMOutCounter.lrTotalCounterEnergy_Production;
END_IF

(*----------------------------------------------------------Save persistent data----------------------------------------------------------------*)

fbPD(lrValue:= BOOL_TO_LREAL(bEnable), bEventBasedActive=> );

END_FUNCTION_BLOCK

// ---- FBs/Meter/M_Bus/Electric/Optec/FB_EM_Optec_Electric_3P.TcPOU
FUNCTION_BLOCK FB_EM_Optec_Electric_3P
VAR_INPUT PERSISTENT
	bEnable							: BOOL;											//Enable the function
	usiPrimAddress					: USINT;										//Primary Address from the Meter
	iTimeReadOutInterval			: INT := 900;									//Delay in seconds to read out the electric meter
	diNrOfMBusMasterLine_IN			: DINT;											//Active Number from the MBus Master Function for using on other functions
END_VAR
VAR_INPUT
END_VAR
VAR_OUTPUT
	stDataEMPower					: ST_ElectricMeter_Output_Power;				//Output structure with Data from Electric Meter (Power Data)
	stDataEMCounter					: ST_ElectricMeter_Output_Counter;				//Output structure with Data from Electric Meter (Counter Data)
	stDataEMPowerRealTime			: ST_ElectricMeter_Output_Power;				//Output structure with Data from Electric Meter (Power Data RealTime)
	stDataEMCounterRealTime			: ST_ElectricMeter_Output_Counter;				//Output structure with Data from Electric Meter (Counter Data RealTime)
	diNrOfEM_OUT					: DINT;											//Active Number from the Electric Meter for using on other functions
END_VAR
VAR
	{attribute 'conditionalshow'}
	fbEM							: FB_ElectricMeter;								//Electric Meter Function
	{attribute 'hide'}
	fbNumberDevice					: FB_NumberOfDevice;							//Function block to calcualte the number of the Device
	{attribute 'hide'}
	fbMBusGeneral					: FB_MBUS_General;								//M-Bus Function
	{attribute 'hide'}
	timDissableFunctions			: TON;											//Timer to dissable the Function after Lynus_Standards.Constants_General.tTimeDissableLynusFunctions Days without connection to the Lynus Cloud
	{attribute 'hide'}
	timResetConnectionOnGVL			: TON;											//Timer to try reset the connection Flag on the GVL. (When somebody delete the Connection Function and make only a onlinechange)
	{attribute 'hide'}
	arrPD							: ARRAY[1..4] OF FB_PersistentData_Number;		//Function to save persistent data
	{attribute 'hide'}
	bErrorMbus						: BOOL;											//Error from the M-Bus Function
	{attribute 'hide'}
	byWaitInStep					: BYTE;											//Wait in Step before start to clean data on PLC
	{attribute 'hide'}
	iStateGVLData					: INT;											//State machine to handle the data on the GVL
	{attribute 'hide'}
	diCounterForGVL					: DINT;											//Counter to clean old data on GVL
END_VAR

//Creator : Kai Ebensperger
//Company : Lynus AG
//Date : 30.08.2021
//Version : 1.0.0.0

//With this function block its possible to read out a Electric Meter from the Factory Optec.
//This Function Block read out the Default Values from the Electric Meter. He didn't change the read out Format.
//This function can only be used for 3-phase meters. (_3P)
//This Function block support only Primary Adress Mode.
//Version according to which was implemented : 2.1
//This Function not send the SND_NKE Telegramm and support only the default firt Telegramm from the Meter

//NOTE for diNr.....Designation => 
//_IN = Here Data come in from other Functions or go out to other functions about the GVL
//_OUT = Here Data go out to other functions about the GVL

(*------------------------------------------------------------Limits----------------------------------------------------------------------------------*)

iTimeReadOutInterval := LIMIT(1,iTimeReadOutInterval,3600);
	diNrOfMBusMasterLine_IN := LIMIT(0,diNrOfMBusMasterLine_IN,Constants_Bussystems.diMaxNumberOfMBusMasterKL6781);
		usiPrimAddress := LIMIT(0,usiPrimAddress,250);

(*-------------------------------------------------------------Calcualte the number of EM---------------------------------------------------------------*)

fbNumberDevice(
	diActualNumberOfDevices:= Lynus_Standards.GVL_Energy.stNumberOfDevices.diNumberOfElectricMeters, 
	diMaxNumberOfDevices:= Constants_Energy.diMaxNumberOfElectricMeters, 
	udiCounterOnlineChange:= TwinCAT_SystemInfoVarList._AppInfo.OnlineChangeCnt, 
	bNumberIsCalculatet=> , 
	bFPNumberIsCalculatet=> , 
	bOnlineChange=> , 
	diNumberForThisDevice=> diNrOfEM_OUT, 
	diNumberOfTotalDevices=> );

//Write new Numer on GVL
IF fbNumberDevice.bFPNumberIsCalculatet THEN
	Lynus_Standards.GVL_Energy.stNumberOfDevices.diNumberOfElectricMeters := fbNumberDevice.diNumberOfTotalDevices;	
END_IF

//Delete old Number on GVL
IF fbNumberDevice.bOnlineChange THEN 
	Lynus_Standards.GVL_Energy.stNumberOfDevices.diNumberOfElectricMeters := diNrOfEM_OUT;	
		iStateGVLData := 1; 
END_IF

(*-------------------------------------------------------------Service from Backend is ready and check the connection to backen for dissabel/enable Function---------------------------------------------------------------*)

//Try to reset the variable for connection on the GVL. When all is normal then the Lynus Mqtt connection function set this variable to true in the next cycle
//When we have no connection to the backend then after Lynus_Standards.Constants_General.tTimeDissableLynusFunctions days the Function is dissabled with all of his functionalities
timResetConnectionOnGVL(IN:= NOT timResetConnectionOnGVL.Q, PT:= T#1H, Q=> , ET=> );
	IF timResetConnectionOnGVL.Q THEN Lynus_Standards.GVL_Communicator.bStateConnectionToEnableFunctions := FALSE; END_IF
		IF NOT Lynus_Standards.GVL_Communicator.bStateConnectionToEnableFunctions THEN timDissableFunctions.IN := TRUE; ELSE timDissableFunctions.IN := FALSE; END_IF  
			timDissableFunctions(IN:= , PT:= Lynus_Standards.Constants_General.tTimeDissableLynusFunctions, Q=> , ET=> );

(*----------------------------------------------------------------------------------------M-Bus Communication----------------------------------------------------------------------------------------------*)
			
fbMBusGeneral(
	usiAddress:= usiPrimAddress, 
	stSecAdr:= , 
	eBaudrate:= Lynus_Standards.GVL_Bussystems.stDataOfMBusMasterKL6781[diNrOfMBusMasterLine_IN].eBaudrateMBusKL6781, 
	bStart:= fbEM.bReadOutMeter, 
	bSND_NKE:= FALSE, 
	bReadInit:= TRUE, 
	tMinSendTime:= T#0S, 
	usiUnit:= 1, 
	bDisabled:= FALSE, 
	bBusy=> , 
	bReady=> , 
	bError=> , 
	eError=> , 
	dwIdNumber=> , 
	byStatus=> , 
	byGEN=> , 
	byCounter=> , 
	usiRecivedAdr=> , 
	eMedium=> , 
	sMan=> , 
	arrData=> , 
	stCom:= Lynus_Standards.GVL_Bussystems.stDataOfMBusMasterKL6781[diNrOfMBusMasterLine_IN].stDataMBusCommunicationKL6781);

(*----------------------------------------------------------------------------------------Electric Meter Function for Pv----------------------------------------------------------------------------------------------*)

IF fbMBusGeneral.bError THEN bErrorMbus := TRUE; ELSE bErrorMbus := FALSE; END_IF

//Error
IF timDissableFunctions.Q THEN fbEM.bWarning := TRUE; fbEM.iWarningCode := 0; ELSE fbEM.bWarning := FALSE; END_IF 
	IF Lynus_Standards.GVL_Energy.stNumberOfDevices.diNumberOfElectricMeters > Constants_Energy.diMaxNumberOfElectricMeters OR bErrorMbus THEN fbEM.bError := TRUE; ELSE fbEM.bError := FALSE; END_IF
		IF Lynus_Standards.GVL_Energy.stNumberOfDevices.diNumberOfElectricMeters > Constants_Energy.diMaxNumberOfElectricMeters THEN fbEM.iErrorCode := 1;
		ELSIF bErrorMbus THEN fbEM.iErrorCode := 0;
		END_IF

//Function
fbEM(
	bEnable:= bEnable AND NOT timDissableFunctions.Q, 
	bError:= , 
	bEnableReadOutFunction:= TRUE, 
	bWriteWithDelay:= TRUE, 
	bPowerDataInvers:= TRUE,
	bReadOutDataDone:= fbMBusGeneral.bBusy,
	iTimeReadOutInterval:= iTimeReadOutInterval, 
	iErrorCode:= , 
	iWarningCode:= , 
	lrTotalCounterEnergy_Consumption:= STRING_TO_LREAL(fbMBusGeneral.arrData[7].sValue) + STRING_TO_LREAL(fbMBusGeneral.arrData[11].sValue), 
	lrTotalCounterEnergy_Production:= 0, 
	lrCounterEnergyT1_Consumption:= STRING_TO_LREAL(fbMBusGeneral.arrData[7].sValue), 
	lrCounterEnergyT2_Consumption:= STRING_TO_LREAL(fbMBusGeneral.arrData[11].sValue), 
	lrCounterEnergyT1_Production:= 0, 
	lrCounterEnergyT2_Production:= 0, 
	lrCurrentL1:= STRING_TO_LREAL(fbMBusGeneral.arrData[25].sValue), 
	lrVoltageL1N:= STRING_TO_LREAL(fbMBusGeneral.arrData[22].sValue), 
	lrVoltageL1L2:= 0, 
	lrPowerL1:= STRING_TO_LREAL(fbMBusGeneral.arrData[14].sValue) * 1000, 
	lrCurrentL2:= STRING_TO_LREAL(fbMBusGeneral.arrData[26].sValue), 
	lrVoltageL2N:= STRING_TO_LREAL(fbMBusGeneral.arrData[23].sValue), 
	lrVoltageL2L3:= 0, 
	lrPowerL2:= STRING_TO_LREAL(fbMBusGeneral.arrData[15].sValue) * 1000, 
	lrCurrentL3:= STRING_TO_LREAL(fbMBusGeneral.arrData[27].sValue), 
	lrVoltageL3N:= STRING_TO_LREAL(fbMBusGeneral.arrData[24].sValue), 
	lrVoltageL3L1:= 0, 
	lrPowerL3:= STRING_TO_LREAL(fbMBusGeneral.arrData[16].sValue) * 1000, 
	lrPowerTotal:= fbEM.lrPowerL1 + fbEM.lrPowerL2 + fbEM.lrPowerL3, 
	lrFrequency:= 0, 
	lrReactivePowerTotal:= STRING_TO_LREAL(fbMBusGeneral.arrData[18].sValue) * 1000 + STRING_TO_LREAL(fbMBusGeneral.arrData[19].sValue) * 1000 + STRING_TO_LREAL(fbMBusGeneral.arrData[20].sValue) * 1000, 
	lrApparentPowerTotal:= 0, 
	tTimDelayOutput:= T#5S, 
	stDataEMOutPower=> stDataEMPowerRealTime, 
	stDataEMOutPowerDelay=> stDataEMPower, 
	stDataEMOutCounter=> stDataEMCounterRealTime,
	stDataEMOutCounterDelay=> stDataEMCounter,
	bReadOutMeter=> );
	
(*-----------------------------------------------------------Handle data to Global structure for Electric Meter-----------------------------------------------------------------*)

CASE iStateGVLData OF
	
	0://Init Step
		byWaitInStep := 0;
			diCounterForGVL := 1;
	
	1://Wait for 4 Steps before clean al Data on GVL
		byWaitInStep := byWaitInStep + 1;
			IF byWaitInStep >= 4 AND fbNumberDevice.bNumberIsCalculatet THEN iStateGVLData := 2; END_IF
				//To much Devices, back to the Init step
				IF byWaitInStep >= 4 AND NOT fbNumberDevice.bNumberIsCalculatet THEN iStateGVLData := 0; END_IF	
			
	2://Clear all Data in GVL
		Lynus_Standards.GVL_Energy.stDataElectricMeters[diCounterForGVL].bEnabled := FALSE;	
			Lynus_Standards.GVL_Energy.stDataElectricMeters[diCounterForGVL].byErrorWarning := 0;
				Lynus_Standards.GVL_Energy.stDataElectricMeters[diCounterForGVL].lrCounterEnergyT1_Consumption := 0;
					Lynus_Standards.GVL_Energy.stDataElectricMeters[diCounterForGVL].lrCounterEnergyT1_Production := 0;
						Lynus_Standards.GVL_Energy.stDataElectricMeters[diCounterForGVL].lrCounterEnergyT2_Consumption := 0;
							Lynus_Standards.GVL_Energy.stDataElectricMeters[diCounterForGVL].lrCounterEnergyT2_Production := 0;
								Lynus_Standards.GVL_Energy.stDataElectricMeters[diCounterForGVL].lrPower := 0;
									Lynus_Standards.GVL_Energy.stDataElectricMeters[diCounterForGVL].lrPowerConsumption := 0;
										Lynus_Standards.GVL_Energy.stDataElectricMeters[diCounterForGVL].lrPowerProduction := 0;
											Lynus_Standards.GVL_Energy.stDataElectricMeters[diCounterForGVL].lrTotalCounterEnergy_Consumption := 0;
												Lynus_Standards.GVL_Energy.stDataElectricMeters[diCounterForGVL].lrTotalCounterEnergy_Production := 0;
		
		//Electric Meters
		diCounterForGVL := diCounterForGVL + 1;
			diCounterForGVL := LIMIT(0,diCounterForGVL,Constants_Energy.diMaxNumberOfElectricMeters);
				//Back to the init step
				IF diCounterForGVL >= Constants_Energy.diMaxNumberOfElectricMeters THEN iStateGVLData := 0; END_IF

END_CASE 	 

//Write Data on GVL for Electric Meter
IF diNrOfEM_OUT > 0 AND fbNumberDevice.bNumberIsCalculatet THEN
	Lynus_Standards.GVL_Energy.stDataElectricMeters[diNrOfEM_OUT].bEnabled := fbEM.stDataEMOutPower.bEnabled;
		Lynus_Standards.GVL_Energy.stDataElectricMeters[diNrOfEM_OUT].byErrorWarning := fbEM.stDataEMOutPower.byErrorWarning;
			Lynus_Standards.GVL_Energy.stDataElectricMeters[diNrOfEM_OUT].lrCounterEnergyT1_Consumption := fbEM.stDataEMOutCounter.lrCounterEnergyT1_Consumption;
				Lynus_Standards.GVL_Energy.stDataElectricMeters[diNrOfEM_OUT].lrCounterEnergyT1_Production := fbEM.stDataEMOutCounter.lrCounterEnergyT1_Production;
					Lynus_Standards.GVL_Energy.stDataElectricMeters[diNrOfEM_OUT].lrCounterEnergyT2_Consumption := fbEM.stDataEMOutCounter.lrCounterEnergyT2_Consumption;
						Lynus_Standards.GVL_Energy.stDataElectricMeters[diNrOfEM_OUT].lrCounterEnergyT2_Production := fbEM.stDataEMOutCounter.lrCounterEnergyT2_Production;		
							Lynus_Standards.GVL_Energy.stDataElectricMeters[diNrOfEM_OUT].lrPower := fbEM.stDataEMOutPower.lrPowerTotal;
								Lynus_Standards.GVL_Energy.stDataElectricMeters[diNrOfEM_OUT].lrPowerConsumption := fbEM.stDataEMOutPower.lrPowerConsumption;
									Lynus_Standards.GVL_Energy.stDataElectricMeters[diNrOfEM_OUT].lrPowerProduction := fbEM.stDataEMOutPower.lrPowerProduction;
										Lynus_Standards.GVL_Energy.stDataElectricMeters[diNrOfEM_OUT].lrTotalCounterEnergy_Consumption := fbEM.stDataEMOutCounter.lrTotalCounterEnergy_Consumption;
											Lynus_Standards.GVL_Energy.stDataElectricMeters[diNrOfEM_OUT].lrTotalCounterEnergy_Production := fbEM.stDataEMOutCounter.lrTotalCounterEnergy_Production;
END_IF

(*----------------------------------------------------------Save persistent data----------------------------------------------------------------*)

arrPD[1](lrValue:= BOOL_TO_LREAL(bEnable), bEventBasedActive=> );
arrPD[2](lrValue:= INT_TO_LREAL(iTimeReadOutInterval), bEventBasedActive=> );
arrPD[3](lrValue:= USINT_TO_LREAL(usiPrimAddress), bEventBasedActive=> );
arrPD[4](lrValue:= DINT_TO_LREAL(diNrOfMBusMasterLine_IN), bEventBasedActive=> );

END_FUNCTION_BLOCK

